LIN {X 0,Y 331.873,Z 625.786,A -85,B 0,C 180,E1 -14668.787,E2 -14668.787} C_VEL
LIN {X 0,Y 331.873,Z 625.82,A -85,B 0,C 180,E1 -14671.213,E2 -14671.213} C_VEL
LIN {X 0,Y 332.002,Z 624.514,A -85,B 0,C 180,E1 -14673.641,E2 -14673.641} C_VEL
LIN {X 0,Y 332.144,Z 621.851,A -85,B 0,C 180,E1 -14676.073,E2 -14676.073} C_VEL
LIN {X 0,Y 332.562,Z 617.761,A -85,B 0,C 180,E1 -14678.507,E2 -14678.507} C_VEL
LIN {X 0,Y 333.251,Z 612.118,A -85,B 0,C 180,E1 -14680.941,E2 -14680.941} C_VEL
LIN {X 0,Y 334.263,Z 605.737,A -85,B 0,C 180,E1 -14683.063,E2 -14683.063} C_VEL
LIN {X 0,Y 335.336,Z 598.598,A -85,B 0,C 180,E1 -14684.985,E2 -14684.985} C_VEL
LIN {X 0,Y 336.771,Z 589.501,A -85,B 0,C 180,E1 -14686.988,E2 -14686.988} C_VEL
LIN {X 0,Y 338.406,Z 579.466,A -85,B 0,C 180,E1 -14688.778,E2 -14688.778} C_VEL
LIN {X 0,Y 340.141,Z 568.232,A -85,B 0,C 180,E1 -14690.406,E2 -14690.406} C_VEL
LIN {X 0,Y 342.003,Z 555.922,A -85,B 0,C 180,E1 -14691.84,E2 -14691.84} C_VEL
LIN {X 0,Y 343.496,Z 543.513,A -85,B 0,C 180,E1 -14693.005,E2 -14693.005} C_VEL
LIN {X 0,Y 344.422,Z 532.816,A -85,B 0,C 180,E1 -14693.822,E2 -14693.822} C_VEL
LIN {X 0,Y 342.468,Z 519.71,A -85,B 0,C 180,E1 -14694.821,E2 -14694.821} C_VEL
LIN {X 0,Y 339.384,Z 505.28,A -85,B 0,C 180,E1 -14695.737,E2 -14695.737} C_VEL
LIN {X 0,Y 335.483,Z 491.266,A -85,B 0,C 180,E1 -14696.482,E2 -14696.482} C_VEL
LIN {X 0,Y 336.062,Z 480.841,A -85,B 0,C 180,E1 -14700.126,E2 -14700.126} C_VEL
LIN {X 0,Y 336.692,Z 470.956,A -85,B 0,C 180,E1 -14703.749,E2 -14703.749} C_VEL
LIN {X 0,Y 337.429,Z 460.368,A -85,B 0,C 180,E1 -14707.725,E2 -14707.725} C_VEL
LIN {X 0,Y 337.849,Z 455.305,A -85,B 0,C 180,E1 -14709.674,E2 -14709.674} C_VEL
LIN {X 0,Y 337.284,Z 449.99,A -85,B 0,C 180,E1 -14711.82,E2 -14711.82} C_VEL
LIN {X 0,Y 337.024,Z 448.414,A -85,B 0,C 180,E1 -14712.464,E2 -14712.464} C_VEL
LIN {X 0,Y 335.911,Z 446.445,A -85,B 0,C 180,E1 -14713.393,E2 -14713.393} C_VEL
LIN {X 0,Y 332.443,Z 443.786,A -85,B 0,C 180,E1 -14714.92,E2 -14714.92} C_VEL
LIN {X 0,Y 329.565,Z 441.699,A -85,B 0,C 180,E1 -14716.158,E2 -14716.158} C_VEL
LIN {X 0,Y 328.141,Z 439.808,A -85,B 0,C 180,E1 -14717.112,E2 -14717.112} C_VEL
LIN {X 0,Y 327.913,Z 439.09,A -85,B 0,C 180,E1 -14717.433,E2 -14717.433} C_VEL
LIN {X 0,Y 326.575,Z 433.434,A -85,B 0,C 180,E1 -14719.993,E2 -14719.993} C_VEL
LIN {X 0,Y 326.632,Z 433.419,A -85,B 0,C 180,E1 -14722.953,E2 -14722.953} C_VEL
LIN {X 0,Y 326.608,Z 433.417,A -85,B 0,C 180,E1 -14725.981,E2 -14725.981} C_VEL
LIN {X 0,Y 326.662,Z 433.41,A -85,B 0,C 180,E1 -14730.341,E2 -14730.341} C_VEL
LIN {X 0,Y 326.723,Z 433.414,A -85,B 0,C 180,E1 -14732.753,E2 -14732.753} C_VEL
LIN {X 0,Y 331.867,Z 449.308,A -85,B 0,C 180,E1 -14734.256,E2 -14734.256} C_VEL
LIN {X 0,Y 336.117,Z 463.308,A -85,B 0,C 180,E1 -14735.79,E2 -14735.79} C_VEL
LIN {X 0,Y 334.703,Z 476.843,A -85,B 0,C 180,E1 -14737.207,E2 -14737.207} C_VEL
LIN {X 0,Y 333.158,Z 489.7,A -85,B 0,C 180,E1 -14738.829,E2 -14738.829} C_VEL
LIN {X 0,Y 331.728,Z 500.872,A -85,B 0,C 180,E1 -14740.508,E2 -14740.508} C_VEL
LIN {X 0,Y 330.337,Z 511.243,A -85,B 0,C 180,E1 -14742.352,E2 -14742.352} C_VEL
LIN {X 0,Y 329.006,Z 521.51,A -85,B 0,C 180,E1 -14744.548,E2 -14744.548} C_VEL
LIN {X 0,Y 328.113,Z 528.711,A -85,B 0,C 180,E1 -14746.372,E2 -14746.372} C_VEL
LIN {X 0,Y 327.375,Z 534.919,A -85,B 0,C 180,E1 -14748.232,E2 -14748.232} C_VEL
LIN {X 0,Y 326.657,Z 541.736,A -85,B 0,C 180,E1 -14750.714,E2 -14750.714} C_VEL
LIN {X 0,Y 326.171,Z 547.048,A -85,B 0,C 180,E1 -14753.194,E2 -14753.194} C_VEL
LIN {X 0,Y 326.088,Z 550.153,A -85,B 0,C 180,E1 -14755.054,E2 -14755.054} C_VEL
LIN {X 0,Y 326.037,Z 551.802,A -85,B 0,C 180,E1 -14756.292,E2 -14756.292} C_VEL
LIN {X 0,Y 325.663,Z 554.196,A -85,B 0,C 180,E1 -14758.763,E2 -14758.763} C_VEL
LIN {X 0,Y 325.695,Z 555.343,A -85,B 0,C 180,E1 -14761.236,E2 -14761.236} C_VEL
LIN {X 0,Y 326.126,Z 555.262,A -85,B 0,C 180,E1 -14763.707,E2 -14763.707} C_VEL
LIN {X 0,Y 326.85,Z 553.984,A -85,B 0,C 180,E1 -14766.172,E2 -14766.172} C_VEL
LIN {X 0,Y 327.566,Z 551.529,A -85,B 0,C 180,E1 -14768.638,E2 -14768.638} C_VEL
LIN {X 0,Y 328.631,Z 547.803,A -85,B 0,C 180,E1 -14771.097,E2 -14771.097} C_VEL
LIN {X 0,Y 329.899,Z 542.755,A -85,B 0,C 180,E1 -14773.553,E2 -14773.553} C_VEL
LIN {X 0,Y 331.726,Z 536.167,A -85,B 0,C 180,E1 -14775.987,E2 -14775.987} C_VEL
LIN {X 0,Y 333.332,Z 530.273,A -85,B 0,C 180,E1 -14777.767,E2 -14777.767} C_VEL
LIN {X 0,Y 335.53,Z 521.743,A -85,B 0,C 180,E1 -14779.899,E2 -14779.899} C_VEL
LIN {X 0,Y 337.941,Z 511.714,A -85,B 0,C 180,E1 -14781.983,E2 -14781.983} C_VEL
LIN {X 0,Y 340.369,Z 501.358,A -85,B 0,C 180,E1 -14783.743,E2 -14783.743} C_VEL
LIN {X 0,Y 342.799,Z 490.786,A -85,B 0,C 180,E1 -14785.247,E2 -14785.247} C_VEL
LIN {X 0,Y 345.29,Z 477.829,A -85,B 0,C 180,E1 -14786.809,E2 -14786.809} C_VEL
LIN {X 0,Y 345.923,Z 474.416,A -85,B 0,C 180,E1 -14787.17,E2 -14787.17} C_VEL
LIN {X 0,Y 345.625,Z 471.773,A -85,B 0,C 180,E1 -14787.571,E2 -14787.571} C_VEL
LIN {X 0,Y 342.511,Z 461.947,A -85,B 0,C 180,E1 -14789.341,E2 -14789.341} C_VEL
LIN {X 0,Y 338.653,Z 453.425,A -85,B 0,C 180,E1 -14791.112,E2 -14791.112} C_VEL
LIN {X 0,Y 335.334,Z 447.304,A -85,B 0,C 180,E1 -14792.574,E2 -14792.574} C_VEL
LIN {X 0,Y 332.623,Z 443.026,A -85,B 0,C 180,E1 -14793.782,E2 -14793.782} C_VEL
LIN {X 0,Y 329.74,Z 438.96,A -85,B 0,C 180,E1 -14795.133,E2 -14795.133} C_VEL
LIN {X 0,Y 327.765,Z 437.307,A -85,B 0,C 180,E1 -14796.036,E2 -14796.036} C_VEL
LIN {X 0,Y 327.108,Z 435.891,A -85,B 0,C 180,E1 -14796.502,E2 -14796.502} C_VEL
LIN {X 0,Y 327.676,Z 439.473,A -85,B 0,C 180,E1 -14800.049,E2 -14800.049} C_VEL
LIN {X 0,Y 328.164,Z 442.306,A -85,B 0,C 180,E1 -14802.424,E2 -14802.424} C_VEL
LIN {X 0,Y 328.168,Z 444.668,A -85,B 0,C 180,E1 -14804.157,E2 -14804.157} C_VEL
LIN {X 0,Y 327.273,Z 451.1,A -85,B 0,C 180,E1 -14808.263,E2 -14808.263} C_VEL
LIN {X 0,Y 326.824,Z 457.809,A -85,B 0,C 180,E1 -14812.135,E2 -14812.135} C_VEL
LIN {X 0,Y 326.571,Z 463.902,A -85,B 0,C 180,E1 -14815.413,E2 -14815.413} C_VEL
LIN {X 0,Y 326.57,Z 464.705,A -85,B 0,C 180,E1 -14815.695,E2 -14815.695} C_VEL
LIN {X 0,Y 327.406,Z 468.646,A -85,B 0,C 180,E1 -14816.306,E2 -14816.306} C_VEL
LIN {X 0,Y 329.147,Z 472.574,A -85,B 0,C 180,E1 -14817.115,E2 -14817.115} C_VEL
LIN {X 0,Y 330.081,Z 476.56,A -85,B 0,C 180,E1 -14817.691,E2 -14817.691} C_VEL
LIN {X 0,Y 331.041,Z 478.958,A -85,B 0,C 180,E1 -14818.125,E2 -14818.125} C_VEL
LIN {X 0,Y 332.455,Z 484.387,A -85,B 0,C 180,E1 -14818.908,E2 -14818.908} C_VEL
LIN {X 0,Y 334.889,Z 495.067,A -85,B 0,C 180,E1 -14820.344,E2 -14820.344} C_VEL
LIN {X 0,Y 336.866,Z 508.787,A -85,B 0,C 180,E1 -14821.993,E2 -14821.993} C_VEL
LIN {X 0,Y 337.451,Z 521.179,A -85,B 0,C 180,E1 -14823.4,E2 -14823.4} C_VEL
LIN {X 0,Y 336.728,Z 537.938,A -85,B 0,C 180,E1 -14825.328,E2 -14825.328} C_VEL
LIN {X 0,Y 336.663,Z 546.487,A -85,B 0,C 180,E1 -14826.469,E2 -14826.469} C_VEL
LIN {X 0,Y 335.948,Z 551.732,A -85,B 0,C 180,E1 -14826.961,E2 -14826.961} C_VEL
LIN {X 0,Y 334.463,Z 563.284,A -85,B 0,C 180,E1 -14828.101,E2 -14828.101} C_VEL
LIN {X 0,Y 332.625,Z 575.509,A -85,B 0,C 180,E1 -14829.597,E2 -14829.597} C_VEL
LIN {X 0,Y 331.031,Z 585.559,A -85,B 0,C 180,E1 -14831.109,E2 -14831.109} C_VEL
LIN {X 0,Y 329.359,Z 595.531,A -85,B 0,C 180,E1 -14832.938,E2 -14832.938} C_VEL
LIN {X 0,Y 328.18,Z 603.43,A -85,B 0,C 180,E1 -14834.697,E2 -14834.697} C_VEL
LIN {X 0,Y 326.9,Z 611.673,A -85,B 0,C 180,E1 -14836.954,E2 -14836.954} C_VEL
LIN {X 0,Y 326.037,Z 617.186,A -85,B 0,C 180,E1 -14838.814,E2 -14838.814} C_VEL
LIN {X 0,Y 325.388,Z 622.949,A -85,B 0,C 180,E1 -14841.304,E2 -14841.304} C_VEL
LIN {X 0,Y 325.053,Z 627.131,A -85,B 0,C 180,E1 -14843.794,E2 -14843.794} C_VEL
LIN {X 0,Y 324.937,Z 629.863,A -85,B 0,C 180,E1 -14846.28,E2 -14846.28} C_VEL
LIN {X 0,Y 324.857,Z 631.218,A -85,B 0,C 180,E1 -14848.76,E2 -14848.76} C_VEL
LIN {X 0,Y 324.857,Z 631.216,A -85,B 0,C 180,E1 -14851.24,E2 -14851.24} C_VEL
LIN {X 0,Y 324.932,Z 629.857,A -85,B 0,C 180,E1 -14853.72,E2 -14853.72} C_VEL
LIN {X 0,Y 325.011,Z 627.122,A -85,B 0,C 180,E1 -14856.207,E2 -14856.207} C_VEL
LIN {X 0,Y 325.382,Z 622.931,A -85,B 0,C 180,E1 -14858.696,E2 -14858.696} C_VEL
LIN {X 0,Y 326.029,Z 617.159,A -85,B 0,C 180,E1 -14861.187,E2 -14861.187} C_VEL
LIN {X 0,Y 327.059,Z 610.636,A -85,B 0,C 180,E1 -14863.356,E2 -14863.356} C_VEL
LIN {X 0,Y 328.14,Z 602.769,A -85,B 0,C 180,E1 -14865.464,E2 -14865.464} C_VEL
LIN {X 0,Y 329.609,Z 593.978,A -85,B 0,C 180,E1 -14867.368,E2 -14867.368} C_VEL
LIN {X 0,Y 331.256,Z 583.611,A -85,B 0,C 180,E1 -14869.199,E2 -14869.199} C_VEL
LIN {X 0,Y 332.951,Z 573.163,A -85,B 0,C 180,E1 -14870.705,E2 -14870.705} C_VEL
LIN {X 0,Y 334.638,Z 561.769,A -85,B 0,C 180,E1 -14872.049,E2 -14872.049} C_VEL
LIN {X 0,Y 336.113,Z 549.889,A -85,B 0,C 180,E1 -14873.186,E2 -14873.186} C_VEL
LIN {X 0,Y 336.405,Z 544.502,A -85,B 0,C 180,E1 -14873.647,E2 -14873.647} C_VEL
LIN {X 0,Y 334.969,Z 531.463,A -85,B 0,C 180,E1 -14874.731,E2 -14874.731} C_VEL
LIN {X 0,Y 332.626,Z 516.987,A -85,B 0,C 180,E1 -14875.72,E2 -14875.72} C_VEL
LIN {X 0,Y 329.791,Z 502.321,A -85,B 0,C 180,E1 -14876.487,E2 -14876.487} C_VEL
LIN {X 0,Y 326.806,Z 490.048,A -85,B 0,C 180,E1 -14877.048,E2 -14877.048} C_VEL
LIN {X 0,Y 326.391,Z 486.716,A -85,B 0,C 180,E1 -14877.491,E2 -14877.491} C_VEL
LIN {X 0,Y 326.933,Z 480.059,A -85,B 0,C 180,E1 -14881.059,E2 -14881.059} C_VEL
LIN {X 0,Y 327.472,Z 473.478,A -85,B 0,C 180,E1 -14884.646,E2 -14884.646} C_VEL
LIN {X 0,Y 327.976,Z 466.679,A -85,B 0,C 180,E1 -14888.42,E2 -14888.42} C_VEL
LIN {X 0,Y 328.616,Z 459.795,A -85,B 0,C 180,E1 -14892.352,E2 -14892.352} C_VEL
LIN {X 0,Y 329.189,Z 453.882,A -85,B 0,C 180,E1 -14895.805,E2 -14895.805} C_VEL
LIN {X 0,Y 329.373,Z 449.755,A -85,B 0,C 180,E1 -14898.315,E2 -14898.315} C_VEL
LIN {X 0,Y 328.587,Z 444.529,A -85,B 0,C 180,E1 -14901.664,E2 -14901.664} C_VEL
LIN {X 0,Y 327.61,Z 439.041,A -85,B 0,C 180,E1 -14905.355,E2 -14905.355} C_VEL
LIN {X 0,Y 326.68,Z 433.42,A -85,B 0,C 180,E1 -14909.377,E2 -14909.377} C_VEL
LIN {X 0,Y 326.686,Z 433.404,A -85,B 0,C 180,E1 -14913.143,E2 -14913.143} C_VEL
LIN {X 0,Y 326.653,Z 433.419,A -85,B 0,C 180,E1 -14915.871,E2 -14915.871} C_VEL
LIN {X 0,Y 326.666,Z 433.402,A -85,B 0,C 180,E1 -14919.865,E2 -14919.865} C_VEL
LIN {X 0,Y 326.701,Z 433.415,A -85,B 0,C 180,E1 -14922.472,E2 -14922.472} C_VEL
LIN {X 0,Y 326.761,Z 433.396,A -85,B 0,C 180,E1 -14926.315,E2 -14926.315} C_VEL
LIN {X 0,Y 326.785,Z 433.391,A -85,B 0,C 180,E1 -14930.093,E2 -14930.093} C_VEL
LIN {X 0,Y 326.985,Z 433.38,A -85,B 0,C 180,E1 -14933.831,E2 -14933.831} C_VEL
LIN {X 0,Y 327.048,Z 433.354,A -85,B 0,C 180,E1 -14937.537,E2 -14937.537} C_VEL
LIN {X 0,Y 327.219,Z 433.353,A -85,B 0,C 180,E1 -14940,E2 -14940} C_VEL
LIN {X 0,Y 327.047,Z 433.356,A -85,B 0,C 180,E1 -14942.463,E2 -14942.463} C_VEL
LIN {X 0,Y 326.973,Z 433.375,A -85,B 0,C 180,E1 -14946.665,E2 -14946.665} C_VEL
LIN {X 0,Y 326.816,Z 433.394,A -85,B 0,C 180,E1 -14949.906,E2 -14949.906} C_VEL
LIN {X 0,Y 326.761,Z 433.394,A -85,B 0,C 180,E1 -14953.685,E2 -14953.685} C_VEL
LIN {X 0,Y 326.701,Z 433.41,A -85,B 0,C 180,E1 -14957.528,E2 -14957.528} C_VEL
LIN {X 0,Y 326.66,Z 433.42,A -85,B 0,C 180,E1 -14960.135,E2 -14960.135} C_VEL
LIN {X 0,Y 326.651,Z 433.418,A -85,B 0,C 180,E1 -14964.129,E2 -14964.129} C_VEL
LIN {X 0,Y 326.686,Z 433.408,A -85,B 0,C 180,E1 -14966.858,E2 -14966.858} C_VEL
LIN {X 0,Y 326.64,Z 433.418,A -85,B 0,C 180,E1 -14970.611,E2 -14970.611} C_VEL
LIN {X 0,Y 326.608,Z 433.427,A -85,B 0,C 180,E1 -14974.019,E2 -14974.019} C_VEL
LIN {X 0,Y 326.629,Z 433.424,A -85,B 0,C 180,E1 -14977.239,E2 -14977.239} C_VEL
LIN {X 0,Y 326.591,Z 433.465,A -85,B 0,C 180,E1 -14980.209,E2 -14980.209} C_VEL
LIN {X 0,Y 328.202,Z 440.412,A -85,B 0,C 180,E1 -14983.276,E2 -14983.276} C_VEL
LIN {X 0,Y 329.71,Z 447.69,A -85,B 0,C 180,E1 -14986.447,E2 -14986.447} C_VEL
LIN {X 0,Y 330.874,Z 454.772,A -85,B 0,C 180,E1 -14989.421,E2 -14989.421} C_VEL
LIN {X 0,Y 330.831,Z 459.25,A -85,B 0,C 180,E1 -14991.195,E2 -14991.195} C_VEL
LIN {X 0,Y 330.039,Z 468.945,A -85,B 0,C 180,E1 -14994.904,E2 -14994.904} C_VEL
LIN {X 0,Y 329.393,Z 478.804,A -85,B 0,C 180,E1 -14998.589,E2 -14998.589} C_VEL
LIN {X 0,Y 328.709,Z 489.231,A -85,B 0,C 180,E1 -15002.323,E2 -15002.323} C_VEL
LIN {X 0,Y 328.622,Z 491.3,A -85,B 0,C 180,E1 -15003.043,E2 -15003.043} C_VEL
LIN {X 0,Y 333.181,Z 507.767,A -85,B 0,C 180,E1 -15003.955,E2 -15003.955} C_VEL
LIN {X 0,Y 335.987,Z 521.344,A -85,B 0,C 180,E1 -15004.867,E2 -15004.867} C_VEL
LIN {X 0,Y 337.83,Z 534.358,A -85,B 0,C 180,E1 -15005.904,E2 -15005.904} C_VEL
LIN {X 0,Y 336.477,Z 547.218,A -85,B 0,C 180,E1 -15006.942,E2 -15006.942} C_VEL
LIN {X 0,Y 334.927,Z 558.972,A -85,B 0,C 180,E1 -15008.133,E2 -15008.133} C_VEL
LIN {X 0,Y 333.02,Z 570.868,A -85,B 0,C 180,E1 -15009.622,E2 -15009.622} C_VEL
LIN {X 0,Y 331.469,Z 580.723,A -85,B 0,C 180,E1 -15011.135,E2 -15011.135} C_VEL
LIN {X 0,Y 329.748,Z 590.533,A -85,B 0,C 180,E1 -15012.959,E2 -15012.959} C_VEL
LIN {X 0,Y 328.425,Z 598.615,A -85,B 0,C 180,E1 -15014.787,E2 -15014.787} C_VEL
LIN {X 0,Y 327.375,Z 605.463,A -85,B 0,C 180,E1 -15016.657,E2 -15016.657} C_VEL
LIN {X 0,Y 326.307,Z 611.907,A -85,B 0,C 180,E1 -15018.823,E2 -15018.823} C_VEL
LIN {X 0,Y 325.516,Z 617.615,A -85,B 0,C 180,E1 -15021.307,E2 -15021.307} C_VEL
LIN {X 0,Y 325.112,Z 621.765,A -85,B 0,C 180,E1 -15023.795,E2 -15023.795} C_VEL
LIN {X 0,Y 324.911,Z 624.482,A -85,B 0,C 180,E1 -15026.279,E2 -15026.279} C_VEL
LIN {X 0,Y 324.785,Z 625.845,A -85,B 0,C 180,E1 -15028.76,E2 -15028.76} C_VEL
LIN {X 0,Y 324.785,Z 625.878,A -85,B 0,C 180,E1 -15031.24,E2 -15031.24} C_VEL
LIN {X 0,Y 324.909,Z 624.572,A -85,B 0,C 180,E1 -15033.721,E2 -15033.721} C_VEL
LIN {X 0,Y 325.078,Z 621.908,A -85,B 0,C 180,E1 -15036.206,E2 -15036.206} C_VEL
LIN {X 0,Y 325.513,Z 617.818,A -85,B 0,C 180,E1 -15038.693,E2 -15038.693} C_VEL
LIN {X 0,Y 326.252,Z 612.173,A -85,B 0,C 180,E1 -15041.179,E2 -15041.179} C_VEL
LIN {X 0,Y 327.332,Z 605.791,A -85,B 0,C 180,E1 -15043.345,E2 -15043.345} C_VEL
LIN {X 0,Y 328.407,Z 598.891,A -85,B 0,C 180,E1 -15045.246,E2 -15045.246} C_VEL
LIN {X 0,Y 329.959,Z 589.552,A -85,B 0,C 180,E1 -15047.349,E2 -15047.349} C_VEL
LIN {X 0,Y 331.674,Z 579.513,A -85,B 0,C 180,E1 -15049.174,E2 -15049.174} C_VEL
LIN {X 0,Y 333.49,Z 568.275,A -85,B 0,C 180,E1 -15050.832,E2 -15050.832} C_VEL
LIN {X 0,Y 335.406,Z 556.051,A -85,B 0,C 180,E1 -15052.281,E2 -15052.281} C_VEL
LIN {X 0,Y 336.993,Z 543.216,A -85,B 0,C 180,E1 -15053.506,E2 -15053.506} C_VEL
LIN {X 0,Y 337.882,Z 534.69,A -85,B 0,C 180,E1 -15054.174,E2 -15054.174} C_VEL
LIN {X 0,Y 336.07,Z 521.646,A -85,B 0,C 180,E1 -15055.217,E2 -15055.217} C_VEL
LIN {X 0,Y 333.145,Z 507.533,A -85,B 0,C 180,E1 -15056.165,E2 -15056.165} C_VEL
LIN {X 0,Y 328.615,Z 491.257,A -85,B 0,C 180,E1 -15057.082,E2 -15057.082} C_VEL
LIN {X 0,Y 329.268,Z 480.763,A -85,B 0,C 180,E1 -15060.815,E2 -15060.815} C_VEL
LIN {X 0,Y 329.91,Z 471.177,A -85,B 0,C 180,E1 -15064.369,E2 -15064.369} C_VEL
LIN {X 0,Y 330.635,Z 461.278,A -85,B 0,C 180,E1 -15068.142,E2 -15068.142} C_VEL
LIN {X 0,Y 330.991,Z 456.139,A -85,B 0,C 180,E1 -15070.146,E2 -15070.146} C_VEL
LIN {X 0,Y 330.219,Z 450.389,A -85,B 0,C 180,E1 -15072.539,E2 -15072.539} C_VEL
LIN {X 0,Y 328.665,Z 442.467,A -85,B 0,C 180,E1 -15075.976,E2 -15075.976} C_VEL
LIN {X 0,Y 327.913,Z 439.09,A -85,B 0,C 180,E1 -15077.433,E2 -15077.433} C_VEL
LIN {X 0,Y 326.906,Z 437.972,A -85,B 0,C 180,E1 -15078.065,E2 -15078.065} C_VEL
LIN {X 0,Y 320.343,Z 435.415,A -85,B 0,C 180,E1 -15080.099,E2 -15080.099} C_VEL
LIN {X 0,Y 319.592,Z 434.302,A -85,B 0,C 180,E1 -15080.798,E2 -15080.798} C_VEL
LIN {X 0,Y 319.582,Z 434.304,A -85,B 0,C 180,E1 -15084.457,E2 -15084.457} C_VEL
LIN {X 0,Y 319.534,Z 434.308,A -85,B 0,C 180,E1 -15088.138,E2 -15088.138} C_VEL
LIN {X 0,Y 319.646,Z 434.295,A -85,B 0,C 180,E1 -15091.924,E2 -15091.924} C_VEL
LIN {X 0,Y 319.662,Z 434.293,A -85,B 0,C 180,E1 -15092.359,E2 -15092.359} C_VEL
LIN {X 0,Y 324.546,Z 449.336,A -85,B 0,C 180,E1 -15093.804,E2 -15093.804} C_VEL
LIN {X 0,Y 328.56,Z 462.529,A -85,B 0,C 180,E1 -15095.261,E2 -15095.261} C_VEL
LIN {X 0,Y 329.266,Z 464.876,A -85,B 0,C 180,E1 -15095.543,E2 -15095.543} C_VEL
LIN {X 0,Y 327.815,Z 478.105,A -85,B 0,C 180,E1 -15096.967,E2 -15096.967} C_VEL
LIN {X 0,Y 326.322,Z 490.19,A -85,B 0,C 180,E1 -15098.523,E2 -15098.523} C_VEL
LIN {X 0,Y 324.694,Z 502.333,A -85,B 0,C 180,E1 -15100.397,E2 -15100.397} C_VEL
LIN {X 0,Y 323.285,Z 512.586,A -85,B 0,C 180,E1 -15102.281,E2 -15102.281} C_VEL
LIN {X 0,Y 322.057,Z 521.771,A -85,B 0,C 180,E1 -15104.28,E2 -15104.28} C_VEL
LIN {X 0,Y 321.032,Z 529.91,A -85,B 0,C 180,E1 -15106.388,E2 -15106.388} C_VEL
LIN {X 0,Y 320.184,Z 537.01,A -85,B 0,C 180,E1 -15108.606,E2 -15108.606} C_VEL
LIN {X 0,Y 319.479,Z 543.59,A -85,B 0,C 180,E1 -15111.142,E2 -15111.142} C_VEL
LIN {X 0,Y 319.043,Z 548.682,A -85,B 0,C 180,E1 -15113.676,E2 -15113.676} C_VEL
LIN {X 0,Y 318.972,Z 552.404,A -85,B 0,C 180,E1 -15116.21,E2 -15116.21} C_VEL
LIN {X 0,Y 318.621,Z 554.887,A -85,B 0,C 180,E1 -15118.736,E2 -15118.736} C_VEL
LIN {X 0,Y 318.651,Z 556.143,A -85,B 0,C 180,E1 -15121.264,E2 -15121.264} C_VEL
LIN {X 0,Y 319.104,Z 556.18,A -85,B 0,C 180,E1 -15123.788,E2 -15123.788} C_VEL
LIN {X 0,Y 319.864,Z 555.008,A -85,B 0,C 180,E1 -15126.307,E2 -15126.307} C_VEL
LIN {X 0,Y 320.651,Z 552.676,A -85,B 0,C 180,E1 -15128.825,E2 -15128.825} C_VEL
LIN {X 0,Y 321.788,Z 549.083,A -85,B 0,C 180,E1 -15131.336,E2 -15131.336} C_VEL
LIN {X 0,Y 323.138,Z 544.164,A -85,B 0,C 180,E1 -15133.842,E2 -15133.842} C_VEL
LIN {X 0,Y 325.08,Z 537.764,A -85,B 0,C 180,E1 -15136.323,E2 -15136.323} C_VEL
LIN {X 0,Y 326.812,Z 531.873,A -85,B 0,C 180,E1 -15138.169,E2 -15138.169} C_VEL
LIN {X 0,Y 329.128,Z 523.736,A -85,B 0,C 180,E1 -15140.303,E2 -15140.303} C_VEL
LIN {X 0,Y 331.678,Z 513.904,A -85,B 0,C 180,E1 -15142.421,E2 -15142.421} C_VEL
LIN {X 0,Y 334.25,Z 503.91,A -85,B 0,C 180,E1 -15144.205,E2 -15144.205} C_VEL
LIN {X 0,Y 337.181,Z 491.975,A -85,B 0,C 180,E1 -15145.958,E2 -15145.958} C_VEL
LIN {X 0,Y 339.535,Z 480.884,A -85,B 0,C 180,E1 -15147.343,E2 -15147.343} C_VEL
LIN {X 0,Y 340.297,Z 476.944,A -85,B 0,C 180,E1 -15147.785,E2 -15147.785} C_VEL
LIN {X 0,Y 339.688,Z 473.304,A -85,B 0,C 180,E1 -15148.415,E2 -15148.415} C_VEL
LIN {X 0,Y 337.096,Z 465.108,A -85,B 0,C 180,E1 -15150.024,E2 -15150.024} C_VEL
LIN {X 0,Y 333.288,Z 456.378,A -85,B 0,C 180,E1 -15152.019,E2 -15152.019} C_VEL
LIN {X 0,Y 329.76,Z 449.903,A -85,B 0,C 180,E1 -15153.779,E2 -15153.779} C_VEL
LIN {X 0,Y 326.968,Z 445.59,A -85,B 0,C 180,E1 -15155.235,E2 -15155.235} C_VEL
LIN {X 0,Y 325.259,Z 444.147,A -85,B 0,C 180,E1 -15156.081,E2 -15156.081} C_VEL
LIN {X 0,Y 324.266,Z 442.628,A -85,B 0,C 180,E1 -15156.686,E2 -15156.686} C_VEL
LIN {X 0,Y 322.352,Z 442.114,A -85,B 0,C 180,E1 -15157.623,E2 -15157.623} C_VEL
LIN {X 0,Y 320.756,Z 440.393,A -85,B 0,C 180,E1 -15158.788,E2 -15158.788} C_VEL
LIN {X 0,Y 320.593,Z 439.96,A -85,B 0,C 180,E1 -15159.023,E2 -15159.023} C_VEL
LIN {X 0,Y 321.153,Z 443.19,A -85,B 0,C 180,E1 -15161.923,E2 -15161.923} C_VEL
LIN {X 0,Y 321.126,Z 446.533,A -85,B 0,C 180,E1 -15164.454,E2 -15164.454} C_VEL
LIN {X 0,Y 320.211,Z 453.259,A -85,B 0,C 180,E1 -15168.819,E2 -15168.819} C_VEL
LIN {X 0,Y 319.734,Z 460.23,A -85,B 0,C 180,E1 -15172.901,E2 -15172.901} C_VEL
LIN {X 0,Y 320.468,Z 464.183,A -85,B 0,C 180,E1 -15173.692,E2 -15173.692} C_VEL
LIN {X 0,Y 322.63,Z 469.537,A -85,B 0,C 180,E1 -15175.048,E2 -15175.048} C_VEL
LIN {X 0,Y 323.754,Z 474.413,A -85,B 0,C 180,E1 -15175.904,E2 -15175.904} C_VEL
LIN {X 0,Y 324.916,Z 477.501,A -85,B 0,C 180,E1 -15176.551,E2 -15176.551} C_VEL
LIN {X 0,Y 328.151,Z 490.791,A -85,B 0,C 180,E1 -15178.675,E2 -15178.675} C_VEL
LIN {X 0,Y 330.201,Z 502.399,A -85,B 0,C 180,E1 -15180.292,E2 -15180.292} C_VEL
LIN {X 0,Y 331.337,Z 514.643,A -85,B 0,C 180,E1 -15181.829,E2 -15181.829} C_VEL
LIN {X 0,Y 331.319,Z 525.862,A -85,B 0,C 180,E1 -15183.172,E2 -15183.172} C_VEL
LIN {X 0,Y 330.324,Z 541.724,A -85,B 0,C 180,E1 -15185.153,E2 -15185.153} C_VEL
LIN {X 0,Y 330.235,Z 547.509,A -85,B 0,C 180,E1 -15185.983,E2 -15185.983} C_VEL
LIN {X 0,Y 329.531,Z 550.892,A -85,B 0,C 180,E1 -15186.407,E2 -15186.407} C_VEL
LIN {X 0,Y 327.853,Z 563.245,A -85,B 0,C 180,E1 -15187.636,E2 -15187.636} C_VEL
LIN {X 0,Y 325.962,Z 575.463,A -85,B 0,C 180,E1 -15189.16,E2 -15189.16} C_VEL
LIN {X 0,Y 324.295,Z 585.511,A -85,B 0,C 180,E1 -15190.701,E2 -15190.701} C_VEL
LIN {X 0,Y 322.552,Z 595.48,A -85,B 0,C 180,E1 -15192.567,E2 -15192.567} C_VEL
LIN {X 0,Y 321.209,Z 603.891,A -85,B 0,C 180,E1 -15194.493,E2 -15194.493} C_VEL
LIN {X 0,Y 319.954,Z 611.618,A -85,B 0,C 180,E1 -15196.665,E2 -15196.665} C_VEL
LIN {X 0,Y 319.025,Z 617.13,A -85,B 0,C 180,E1 -15198.564,E2 -15198.564} C_VEL
LIN {X 0,Y 318.347,Z 622.893,A -85,B 0,C 180,E1 -15201.11,E2 -15201.11} C_VEL
LIN {X 0,Y 317.971,Z 627.074,A -85,B 0,C 180,E1 -15203.655,E2 -15203.655} C_VEL
LIN {X 0,Y 317.845,Z 629.805,A -85,B 0,C 180,E1 -15206.197,E2 -15206.197} C_VEL
LIN {X 0,Y 317.768,Z 631.16,A -85,B 0,C 180,E1 -15208.733,E2 -15208.733} C_VEL
LIN {X 0,Y 317.768,Z 631.157,A -85,B 0,C 180,E1 -15211.267,E2 -15211.267} C_VEL
LIN {X 0,Y 317.839,Z 629.799,A -85,B 0,C 180,E1 -15213.804,E2 -15213.804} C_VEL
LIN {X 0,Y 317.951,Z 627.063,A -85,B 0,C 180,E1 -15216.345,E2 -15216.345} C_VEL
LIN {X 0,Y 318.341,Z 622.872,A -85,B 0,C 180,E1 -15218.89,E2 -15218.89} C_VEL
LIN {X 0,Y 319.018,Z 617.101,A -85,B 0,C 180,E1 -15221.436,E2 -15221.436} C_VEL
LIN {X 0,Y 320.121,Z 610.579,A -85,B 0,C 180,E1 -15223.651,E2 -15223.651} C_VEL
LIN {X 0,Y 321.354,Z 602.335,A -85,B 0,C 180,E1 -15225.894,E2 -15225.894} C_VEL
LIN {X 0,Y 322.803,Z 593.922,A -85,B 0,C 180,E1 -15227.746,E2 -15227.746} C_VEL
LIN {X 0,Y 324.54,Z 583.557,A -85,B 0,C 180,E1 -15229.613,E2 -15229.613} C_VEL
LIN {X 0,Y 326.297,Z 573.112,A -85,B 0,C 180,E1 -15231.148,E2 -15231.148} C_VEL
LIN {X 0,Y 328.053,Z 561.721,A -85,B 0,C 180,E1 -15232.516,E2 -15232.516} C_VEL
LIN {X 0,Y 329.564,Z 550.129,A -85,B 0,C 180,E1 -15233.648,E2 -15233.648} C_VEL
LIN {X 0,Y 329.827,Z 546.096,A -85,B 0,C 180,E1 -15234.009,E2 -15234.009} C_VEL
LIN {X 0,Y 328.492,Z 533.124,A -85,B 0,C 180,E1 -15235.142,E2 -15235.142} C_VEL
LIN {X 0,Y 326.242,Z 518.571,A -85,B 0,C 180,E1 -15236.185,E2 -15236.185} C_VEL
LIN {X 0,Y 323.421,Z 503.738,A -85,B 0,C 180,E1 -15237.009,E2 -15237.009} C_VEL
LIN {X 0,Y 320.854,Z 492.766,A -85,B 0,C 180,E1 -15237.527,E2 -15237.527} C_VEL
LIN {X 0,Y 319.931,Z 489.497,A -85,B 0,C 180,E1 -15237.719,E2 -15237.719} C_VEL
LIN {X 0,Y 319.409,Z 485.41,A -85,B 0,C 180,E1 -15238.342,E2 -15238.342} C_VEL
LIN {X 0,Y 319.909,Z 479.077,A -85,B 0,C 180,E1 -15241.82,E2 -15241.82} C_VEL
LIN {X 0,Y 320.411,Z 473.776,A -85,B 0,C 180,E1 -15244.771,E2 -15244.771} C_VEL
LIN {X 0,Y 320.937,Z 467.017,A -85,B 0,C 180,E1 -15248.625,E2 -15248.625} C_VEL
LIN {X 0,Y 321.611,Z 460.087,A -85,B 0,C 180,E1 -15252.643,E2 -15252.643} C_VEL
LIN {X 0,Y 322.195,Z 454.433,A -85,B 0,C 180,E1 -15256.04,E2 -15256.04} C_VEL
LIN {X 0,Y 322.318,Z 450.458,A -85,B 0,C 180,E1 -15258.495,E2 -15258.495} C_VEL
LIN {X 0,Y 321.857,Z 447.033,A -85,B 0,C 180,E1 -15260.711,E2 -15260.711} C_VEL
LIN {X 0,Y 320.942,Z 441.996,A -85,B 0,C 180,E1 -15264.118,E2 -15264.118} C_VEL
LIN {X 0,Y 319.938,Z 436.268,A -85,B 0,C 180,E1 -15268.183,E2 -15268.183} C_VEL
LIN {X 0,Y 319.633,Z 434.299,A -85,B 0,C 180,E1 -15269.712,E2 -15269.712} C_VEL
LIN {X 0,Y 319.636,Z 434.278,A -85,B 0,C 180,E1 -15273.912,E2 -15273.912} C_VEL
LIN {X 0,Y 319.598,Z 434.292,A -85,B 0,C 180,E1 -15278.048,E2 -15278.048} C_VEL
LIN {X 0,Y 319.691,Z 434.282,A -85,B 0,C 180,E1 -15280.962,E2 -15280.962} C_VEL
LIN {X 0,Y 319.732,Z 434.264,A -85,B 0,C 180,E1 -15285.276,E2 -15285.276} C_VEL
LIN {X 0,Y 319.717,Z 434.284,A -85,B 0,C 180,E1 -15288.59,E2 -15288.59} C_VEL
LIN {X 0,Y 319.896,Z 434.252,A -85,B 0,C 180,E1 -15292.425,E2 -15292.425} C_VEL
LIN {X 0,Y 319.746,Z 434.28,A -85,B 0,C 180,E1 -15294.956,E2 -15294.956} C_VEL
LIN {X 0,Y 319.991,Z 434.232,A -85,B 0,C 180,E1 -15297.483,E2 -15297.483} C_VEL
LIN {X 0,Y 320.17,Z 434.231,A -85,B 0,C 180,E1 -15300,E2 -15300} C_VEL
LIN {X 0,Y 319.991,Z 434.234,A -85,B 0,C 180,E1 -15302.518,E2 -15302.518} C_VEL
LIN {X 0,Y 319.933,Z 434.253,A -85,B 0,C 180,E1 -15306.656,E2 -15306.656} C_VEL
LIN {X 0,Y 319.76,Z 434.275,A -85,B 0,C 180,E1 -15310.127,E2 -15310.127} C_VEL
LIN {X 0,Y 319.732,Z 434.274,A -85,B 0,C 180,E1 -15314.724,E2 -15314.724} C_VEL
LIN {X 0,Y 319.69,Z 434.277,A -85,B 0,C 180,E1 -15319.038,E2 -15319.038} C_VEL
LIN {X 0,Y 319.562,Z 434.295,A -85,B 0,C 180,E1 -15323.32,E2 -15323.32} C_VEL
LIN {X 0,Y 319.636,Z 434.289,A -85,B 0,C 180,E1 -15326.088,E2 -15326.088} C_VEL
LIN {X 0,Y 319.591,Z 434.3,A -85,B 0,C 180,E1 -15328.934,E2 -15328.934} C_VEL
LIN {X 0,Y 319.534,Z 434.309,A -85,B 0,C 180,E1 -15331.862,E2 -15331.862} C_VEL
LIN {X 0,Y 319.581,Z 434.298,A -85,B 0,C 180,E1 -15335.543,E2 -15335.543} C_VEL
LIN {X 0,Y 319.576,Z 434.444,A -85,B 0,C 180,E1 -15339.489,E2 -15339.489} C_VEL
LIN {X 0,Y 321.222,Z 441.511,A -85,B 0,C 180,E1 -15342.707,E2 -15342.707} C_VEL
LIN {X 0,Y 322.726,Z 448.775,A -85,B 0,C 180,E1 -15345.943,E2 -15345.943} C_VEL
LIN {X 0,Y 323.834,Z 454.836,A -85,B 0,C 180,E1 -15348.554,E2 -15348.554} C_VEL
LIN {X 0,Y 324.113,Z 458.867,A -85,B 0,C 180,E1 -15350.233,E2 -15350.233} C_VEL
LIN {X 0,Y 323.317,Z 468.701,A -85,B 0,C 180,E1 -15354.062,E2 -15354.062} C_VEL
LIN {X 0,Y 322.614,Z 478.254,A -85,B 0,C 180,E1 -15357.688,E2 -15357.688} C_VEL
LIN {X 0,Y 321.971,Z 488.128,A -85,B 0,C 180,E1 -15361.3,E2 -15361.3} C_VEL
LIN {X 0,Y 321.794,Z 491.392,A -85,B 0,C 180,E1 -15362.432,E2 -15362.432} C_VEL
LIN {X 0,Y 326.317,Z 507.497,A -85,B 0,C 180,E1 -15363.354,E2 -15363.354} C_VEL
LIN {X 0,Y 329.09,Z 520.467,A -85,B 0,C 180,E1 -15364.25,E2 -15364.25} C_VEL
LIN {X 0,Y 331.012,Z 533.387,A -85,B 0,C 180,E1 -15365.298,E2 -15365.298} C_VEL
LIN {X 0,Y 331.135,Z 536.489,A -85,B 0,C 180,E1 -15365.557,E2 -15365.557} C_VEL
LIN {X 0,Y 329.768,Z 548.919,A -85,B 0,C 180,E1 -15366.62,E2 -15366.62} C_VEL
LIN {X 0,Y 327.983,Z 561.558,A -85,B 0,C 180,E1 -15367.976,E2 -15367.976} C_VEL
LIN {X 0,Y 326.007,Z 573.018,A -85,B 0,C 180,E1 -15369.493,E2 -15369.493} C_VEL
LIN {X 0,Y 324.423,Z 582.528,A -85,B 0,C 180,E1 -15371.038,E2 -15371.038} C_VEL
LIN {X 0,Y 322.668,Z 592.051,A -85,B 0,C 180,E1 -15372.9,E2 -15372.9} C_VEL
LIN {X 0,Y 321.336,Z 599.946,A -85,B 0,C 180,E1 -15374.784,E2 -15374.784} C_VEL
LIN {X 0,Y 320.253,Z 606.514,A -85,B 0,C 180,E1 -15376.678,E2 -15376.678} C_VEL
LIN {X 0,Y 319.316,Z 611.966,A -85,B 0,C 180,E1 -15378.575,E2 -15378.575} C_VEL
LIN {X 0,Y 318.482,Z 617.673,A -85,B 0,C 180,E1 -15381.114,E2 -15381.114} C_VEL
LIN {X 0,Y 318.054,Z 621.824,A -85,B 0,C 180,E1 -15383.657,E2 -15383.657} C_VEL
LIN {X 0,Y 317.822,Z 624.541,A -85,B 0,C 180,E1 -15386.196,E2 -15386.196} C_VEL
LIN {X 0,Y 317.699,Z 625.903,A -85,B 0,C 180,E1 -15388.732,E2 -15388.732} C_VEL
LIN {X 0,Y 317.699,Z 625.936,A -85,B 0,C 180,E1 -15391.268,E2 -15391.268} C_VEL
LIN {X 0,Y 317.819,Z 624.63,A -85,B 0,C 180,E1 -15393.804,E2 -15393.804} C_VEL
LIN {X 0,Y 318.012,Z 621.966,A -85,B 0,C 180,E1 -15396.344,E2 -15396.344} C_VEL
LIN {X 0,Y 318.479,Z 617.875,A -85,B 0,C 180,E1 -15398.886,E2 -15398.886} C_VEL
LIN {X 0,Y 319.237,Z 612.229,A -85,B 0,C 180,E1 -15401.428,E2 -15401.428} C_VEL
LIN {X 0,Y 320.38,Z 605.846,A -85,B 0,C 180,E1 -15403.64,E2 -15403.64} C_VEL
LIN {X 0,Y 321.698,Z 598.031,A -85,B 0,C 180,E1 -15405.817,E2 -15405.817} C_VEL
LIN {X 0,Y 323.157,Z 589.603,A -85,B 0,C 180,E1 -15407.726,E2 -15407.726} C_VEL
LIN {X 0,Y 324.957,Z 579.56,A -85,B 0,C 180,E1 -15409.586,E2 -15409.586} C_VEL
LIN {X 0,Y 326.852,Z 568.318,A -85,B 0,C 180,E1 -15411.275,E2 -15411.275} C_VEL
LIN {X 0,Y 328.672,Z 557.146,A -85,B 0,C 180,E1 -15412.637,E2 -15412.637} C_VEL
LIN {X 0,Y 330.261,Z 544.963,A -85,B 0,C 180,E1 -15413.849,E2 -15413.849} C_VEL
LIN {X 0,Y 331.297,Z 535.754,A -85,B 0,C 180,E1 -15414.602,E2 -15414.602} C_VEL
LIN {X 0,Y 329.585,Z 523.164,A -85,B 0,C 180,E1 -15415.658,E2 -15415.658} C_VEL
LIN {X 0,Y 326.722,Z 509.013,A -85,B 0,C 180,E1 -15416.659,E2 -15416.659} C_VEL
LIN {X 0,Y 322.504,Z 493.892,A -85,B 0,C 180,E1 -15417.551,E2 -15417.551} C_VEL
LIN {X 0,Y 321.792,Z 491.276,A -85,B 0,C 180,E1 -15417.696,E2 -15417.696} C_VEL
LIN {X 0,Y 322.336,Z 482.59,A -85,B 0,C 180,E1 -15420.822,E2 -15420.822} C_VEL
LIN {X 0,Y 323.012,Z 472.884,A -85,B 0,C 180,E1 -15424.451,E2 -15424.451} C_VEL
LIN {X 0,Y 323.893,Z 462.065,A -85,B 0,C 180,E1 -15428.634,E2 -15428.634} C_VEL
LIN {X 0,Y 324.11,Z 457.213,A -85,B 0,C 180,E1 -15430.581,E2 -15430.581} C_VEL
LIN {X 0,Y 323.177,Z 451.017,A -85,B 0,C 180,E1 -15433.238,E2 -15433.238} C_VEL
LIN {X 0,Y 321.875,Z 444.487,A -85,B 0,C 180,E1 -15436.099,E2 -15436.099} C_VEL
LIN {X 0,Y 320.095,Z 436.623,A -85,B 0,C 180,E1 -15439.632,E2 -15439.632} C_VEL
LIN {X 0,Y 319.592,Z 434.302,A -85,B 0,C 180,E1 -15440.798,E2 -15440.798} C_VEL
LIN {X 0,Y 318.934,Z 434.388,A -85,B 0,C 180,E1 -15441.85,E2 -15441.85} C_VEL
LIN {X 0,Y 316.101,Z 434.731,A -85,B 0,C 180,E1 -15443.562,E2 -15443.562} C_VEL
LIN {X 0,Y 313.679,Z 435.035,A -85,B 0,C 180,E1 -15444.95,E2 -15444.95} C_VEL
LIN {X 0,Y 312.616,Z 435.16,A -85,B 0,C 180,E1 -15446.024,E2 -15446.024} C_VEL
LIN {X 0,Y 312.516,Z 435.172,A -85,B 0,C 180,E1 -15446.388,E2 -15446.388} C_VEL
LIN {X 0,Y 312.551,Z 435.167,A -85,B 0,C 180,E1 -15450.35,E2 -15450.35} C_VEL
LIN {X 0,Y 312.607,Z 435.201,A -85,B 0,C 180,E1 -15451.955,E2 -15451.955} C_VEL
LIN {X 0,Y 317.245,Z 449.523,A -85,B 0,C 180,E1 -15453.36,E2 -15453.36} C_VEL
LIN {X 0,Y 321.385,Z 462.949,A -85,B 0,C 180,E1 -15454.876,E2 -15454.876} C_VEL
LIN {X 0,Y 322.398,Z 466.614,A -85,B 0,C 180,E1 -15455.323,E2 -15455.323} C_VEL
LIN {X 0,Y 320.864,Z 479.7,A -85,B 0,C 180,E1 -15456.78,E2 -15456.78} C_VEL
LIN {X 0,Y 319.136,Z 492.704,A -85,B 0,C 180,E1 -15458.524,E2 -15458.524} C_VEL
LIN {X 0,Y 317.671,Z 503.681,A -85,B 0,C 180,E1 -15460.282,E2 -15460.282} C_VEL
LIN {X 0,Y 316.207,Z 513.853,A -85,B 0,C 180,E1 -15462.205,E2 -15462.205} C_VEL
LIN {X 0,Y 315.088,Z 522.251,A -85,B 0,C 180,E1 -15464.068,E2 -15464.068} C_VEL
LIN {X 0,Y 314.082,Z 529.931,A -85,B 0,C 180,E1 -15466.081,E2 -15466.081} C_VEL
LIN {X 0,Y 313.191,Z 537.182,A -85,B 0,C 180,E1 -15468.348,E2 -15468.348} C_VEL
LIN {X 0,Y 312.455,Z 543.911,A -85,B 0,C 180,E1 -15470.941,E2 -15470.941} C_VEL
LIN {X 0,Y 311.999,Z 549.127,A -85,B 0,C 180,E1 -15473.533,E2 -15473.533} C_VEL
LIN {X 0,Y 311.912,Z 552.962,A -85,B 0,C 180,E1 -15476.124,E2 -15476.124} C_VEL
LIN {X 0,Y 311.58,Z 555.565,A -85,B 0,C 180,E1 -15478.707,E2 -15478.707} C_VEL
LIN {X 0,Y 311.609,Z 556.945,A -85,B 0,C 180,E1 -15481.292,E2 -15481.292} C_VEL
LIN {X 0,Y 312.083,Z 557.099,A -85,B 0,C 180,E1 -15483.874,E2 -15483.874} C_VEL
LIN {X 0,Y 312.882,Z 556.057,A -85,B 0,C 180,E1 -15486.448,E2 -15486.448} C_VEL
LIN {X 0,Y 313.74,Z 553.845,A -85,B 0,C 180,E1 -15489.021,E2 -15489.021} C_VEL
LIN {X 0,Y 314.963,Z 550.382,A -85,B 0,C 180,E1 -15491.585,E2 -15491.585} C_VEL
LIN {X 0,Y 316.417,Z 545.634,A -85,B 0,C 180,E1 -15494.142,E2 -15494.142} C_VEL
LIN {X 0,Y 318.471,Z 539.381,A -85,B 0,C 180,E1 -15496.671,E2 -15496.671} C_VEL
LIN {X 0,Y 320.324,Z 533.713,A -85,B 0,C 180,E1 -15498.55,E2 -15498.55} C_VEL
LIN {X 0,Y 322.753,Z 525.745,A -85,B 0,C 180,E1 -15500.723,E2 -15500.723} C_VEL
LIN {X 0,Y 325.479,Z 516.239,A -85,B 0,C 180,E1 -15502.872,E2 -15502.872} C_VEL
LIN {X 0,Y 328.665,Z 504.735,A -85,B 0,C 180,E1 -15504.981,E2 -15504.981} C_VEL
LIN {X 0,Y 331.654,Z 493.371,A -85,B 0,C 180,E1 -15506.686,E2 -15506.686} C_VEL
LIN {X 0,Y 334.747,Z 479.83,A -85,B 0,C 180,E1 -15508.404,E2 -15508.404} C_VEL
LIN {X 0,Y 334.324,Z 476.974,A -85,B 0,C 180,E1 -15508.914,E2 -15508.914} C_VEL
LIN {X 0,Y 331.718,Z 468.169,A -85,B 0,C 180,E1 -15510.78,E2 -15510.78} C_VEL
LIN {X 0,Y 327.931,Z 459.193,A -85,B 0,C 180,E1 -15513.062,E2 -15513.062} C_VEL
LIN {X 0,Y 324.195,Z 452.539,A -85,B 0,C 180,E1 -15515.216,E2 -15515.216} C_VEL
LIN {X 0,Y 322.388,Z 450.561,A -85,B 0,C 180,E1 -15516.236,E2 -15516.236} C_VEL
LIN {X 0,Y 319.324,Z 448.352,A -85,B 0,C 180,E1 -15518.043,E2 -15518.043} C_VEL
LIN {X 0,Y 317.773,Z 446.819,A -85,B 0,C 180,E1 -15519.279,E2 -15519.279} C_VEL
LIN {X 0,Y 315.796,Z 446.898,A -85,B 0,C 180,E1 -15520.829,E2 -15520.829} C_VEL
LIN {X 0,Y 314.271,Z 446.522,A -85,B 0,C 180,E1 -15523.373,E2 -15523.373} C_VEL
LIN {X 0,Y 313.725,Z 450.229,A -85,B 0,C 180,E1 -15526.016,E2 -15526.016} C_VEL
LIN {X 0,Y 313.41,Z 453.012,A -85,B 0,C 180,E1 -15527.731,E2 -15527.731} C_VEL
LIN {X 0,Y 314.437,Z 460.638,A -85,B 0,C 180,E1 -15530.454,E2 -15530.454} C_VEL
LIN {X 0,Y 316.423,Z 466.064,A -85,B 0,C 180,E1 -15532.377,E2 -15532.377} C_VEL
LIN {X 0,Y 317.444,Z 471.032,A -85,B 0,C 180,E1 -15533.507,E2 -15533.507} C_VEL
LIN {X 0,Y 318.385,Z 473.666,A -85,B 0,C 180,E1 -15534.206,E2 -15534.206} C_VEL
LIN {X 0,Y 319.934,Z 479.939,A -85,B 0,C 180,E1 -15535.483,E2 -15535.483} C_VEL
LIN {X 0,Y 320.697,Z 482.549,A -85,B 0,C 180,E1 -15536.025,E2 -15536.025} C_VEL
LIN {X 0,Y 323.329,Z 495.236,A -85,B 0,C 180,E1 -15538.177,E2 -15538.177} C_VEL
LIN {X 0,Y 324.956,Z 506.944,A -85,B 0,C 180,E1 -15539.894,E2 -15539.894} C_VEL
LIN {X 0,Y 325.558,Z 518.863,A -85,B 0,C 180,E1 -15541.476,E2 -15541.476} C_VEL
LIN {X 0,Y 325.224,Z 528.408,A -85,B 0,C 180,E1 -15542.689,E2 -15542.689} C_VEL
LIN {X 0,Y 323.992,Z 543,A -85,B 0,C 180,E1 -15544.633,E2 -15544.633} C_VEL
LIN {X 0,Y 323.587,Z 549.639,A -85,B 0,C 180,E1 -15545.628,E2 -15545.628} C_VEL
LIN {X 0,Y 322.609,Z 553.642,A -85,B 0,C 180,E1 -15546.158,E2 -15546.158} C_VEL
LIN {X 0,Y 320.911,Z 565.827,A -85,B 0,C 180,E1 -15547.465,E2 -15547.465} C_VEL
LIN {X 0,Y 318.94,Z 577.549,A -85,B 0,C 180,E1 -15549.018,E2 -15549.018} C_VEL
LIN {X 0,Y 317.233,Z 587.238,A -85,B 0,C 180,E1 -15550.591,E2 -15550.591} C_VEL
LIN {X 0,Y 315.48,Z 596.911,A -85,B 0,C 180,E1 -15552.498,E2 -15552.498} C_VEL
LIN {X 0,Y 314.158,Z 604.915,A -85,B 0,C 180,E1 -15554.428,E2 -15554.428} C_VEL
LIN {X 0,Y 313.024,Z 611.564,A -85,B 0,C 180,E1 -15556.364,E2 -15556.364} C_VEL
LIN {X 0,Y 312.026,Z 617.074,A -85,B 0,C 180,E1 -15558.304,E2 -15558.304} C_VEL
LIN {X 0,Y 311.291,Z 622.836,A -85,B 0,C 180,E1 -15560.907,E2 -15560.907} C_VEL
LIN {X 0,Y 310.9,Z 627.016,A -85,B 0,C 180,E1 -15563.51,E2 -15563.51} C_VEL
LIN {X 0,Y 310.757,Z 629.747,A -85,B 0,C 180,E1 -15566.11,E2 -15566.11} C_VEL
LIN {X 0,Y 310.681,Z 631.102,A -85,B 0,C 180,E1 -15568.704,E2 -15568.704} C_VEL
LIN {X 0,Y 310.681,Z 631.099,A -85,B 0,C 180,E1 -15571.296,E2 -15571.296} C_VEL
LIN {X 0,Y 310.75,Z 629.74,A -85,B 0,C 180,E1 -15573.89,E2 -15573.89} C_VEL
LIN {X 0,Y 310.888,Z 627.005,A -85,B 0,C 180,E1 -15576.49,E2 -15576.49} C_VEL
LIN {X 0,Y 311.28,Z 622.814,A -85,B 0,C 180,E1 -15579.093,E2 -15579.093} C_VEL
LIN {X 0,Y 312.019,Z 617.043,A -85,B 0,C 180,E1 -15581.696,E2 -15581.696} C_VEL
LIN {X 0,Y 313.181,Z 610.521,A -85,B 0,C 180,E1 -15583.96,E2 -15583.96} C_VEL
LIN {X 0,Y 314.434,Z 602.595,A -85,B 0,C 180,E1 -15586.172,E2 -15586.172} C_VEL
LIN {X 0,Y 316.008,Z 593.867,A -85,B 0,C 180,E1 -15588.141,E2 -15588.141} C_VEL
LIN {X 0,Y 317.831,Z 583.504,A -85,B 0,C 180,E1 -15590.044,E2 -15590.044} C_VEL
LIN {X 0,Y 319.662,Z 573.061,A -85,B 0,C 180,E1 -15591.608,E2 -15591.608} C_VEL
LIN {X 0,Y 321.49,Z 561.674,A -85,B 0,C 180,E1 -15593.002,E2 -15593.002} C_VEL
LIN {X 0,Y 323.028,Z 550.354,A -85,B 0,C 180,E1 -15594.131,E2 -15594.131} C_VEL
LIN {X 0,Y 323.069,Z 546.136,A -85,B 0,C 180,E1 -15594.536,E2 -15594.536} C_VEL
LIN {X 0,Y 321.818,Z 533.093,A -85,B 0,C 180,E1 -15595.701,E2 -15595.701} C_VEL
LIN {X 0,Y 319.7,Z 519.109,A -85,B 0,C 180,E1 -15596.736,E2 -15596.736} C_VEL
LIN {X 0,Y 317.013,Z 504.521,A -85,B 0,C 180,E1 -15597.578,E2 -15597.578} C_VEL
LIN {X 0,Y 314.674,Z 494.844,A -85,B 0,C 180,E1 -15598.063,E2 -15598.063} C_VEL
LIN {X 0,Y 313.06,Z 489.426,A -85,B 0,C 180,E1 -15598.402,E2 -15598.402} C_VEL
LIN {X 0,Y 312.477,Z 484.043,A -85,B 0,C 180,E1 -15599.238,E2 -15599.238} C_VEL
LIN {X 0,Y 313.087,Z 476.963,A -85,B 0,C 180,E1 -15603.241,E2 -15603.241} C_VEL
LIN {X 0,Y 313.462,Z 471.867,A -85,B 0,C 180,E1 -15606.182,E2 -15606.182} C_VEL
LIN {X 0,Y 314.026,Z 465.936,A -85,B 0,C 180,E1 -15609.631,E2 -15609.631} C_VEL
LIN {X 0,Y 314.753,Z 458.987,A -85,B 0,C 180,E1 -15613.804,E2 -15613.804} C_VEL
LIN {X 0,Y 315.297,Z 453.212,A -85,B 0,C 180,E1 -15617.356,E2 -15617.356} C_VEL
LIN {X 0,Y 315.053,Z 449.609,A -85,B 0,C 180,E1 -15619.691,E2 -15619.691} C_VEL
LIN {X 0,Y 314.038,Z 443.75,A -85,B 0,C 180,E1 -15623.674,E2 -15623.674} C_VEL
LIN {X 0,Y 313.156,Z 438.506,A -85,B 0,C 180,E1 -15627.41,E2 -15627.41} C_VEL
LIN {X 0,Y 312.585,Z 435.177,A -85,B 0,C 180,E1 -15629.983,E2 -15629.983} C_VEL
LIN {X 0,Y 312.604,Z 435.153,A -85,B 0,C 180,E1 -15634.064,E2 -15634.064} C_VEL
LIN {X 0,Y 312.589,Z 435.169,A -85,B 0,C 180,E1 -15637.529,E2 -15637.529} C_VEL
LIN {X 0,Y 312.64,Z 435.165,A -85,B 0,C 180,E1 -15641.657,E2 -15641.657} C_VEL
LIN {X 0,Y 312.695,Z 435.141,A -85,B 0,C 180,E1 -15645.686,E2 -15645.686} C_VEL
LIN {X 0,Y 312.687,Z 435.152,A -85,B 0,C 180,E1 -15649.641,E2 -15649.641} C_VEL
LIN {X 0,Y 312.895,Z 435.134,A -85,B 0,C 180,E1 -15653.552,E2 -15653.552} C_VEL
LIN {X 0,Y 312.938,Z 435.11,A -85,B 0,C 180,E1 -15657.426,E2 -15657.426} C_VEL
LIN {X 0,Y 313.122,Z 435.109,A -85,B 0,C 180,E1 -15660,E2 -15660} C_VEL
LIN {X 0,Y 312.937,Z 435.111,A -85,B 0,C 180,E1 -15662.574,E2 -15662.574} C_VEL
LIN {X 0,Y 312.896,Z 435.13,A -85,B 0,C 180,E1 -15666.639,E2 -15666.639} C_VEL
LIN {X 0,Y 312.789,Z 435.131,A -85,B 0,C 180,E1 -15669.049,E2 -15669.049} C_VEL
LIN {X 0,Y 312.636,Z 435.156,A -85,B 0,C 180,E1 -15672.991,E2 -15672.991} C_VEL
LIN {X 0,Y 312.64,Z 435.167,A -85,B 0,C 180,E1 -15675.65,E2 -15675.65} C_VEL
LIN {X 0,Y 312.61,Z 435.159,A -85,B 0,C 180,E1 -15679.225,E2 -15679.225} C_VEL
LIN {X 0,Y 312.527,Z 435.17,A -85,B 0,C 180,E1 -15682.781,E2 -15682.781} C_VEL
LIN {X 0,Y 312.604,Z 435.165,A -85,B 0,C 180,E1 -15685.936,E2 -15685.936} C_VEL
LIN {X 0,Y 312.547,Z 435.173,A -85,B 0,C 180,E1 -15689.65,E2 -15689.65} C_VEL
LIN {X 0,Y 312.521,Z 435.178,A -85,B 0,C 180,E1 -15693.689,E2 -15693.689} C_VEL
LIN {X 0,Y 312.527,Z 435.179,A -85,B 0,C 180,E1 -15697.385,E2 -15697.385} C_VEL
LIN {X 0,Y 312.572,Z 435.373,A -85,B 0,C 180,E1 -15698.729,E2 -15698.729} C_VEL
LIN {X 0,Y 314.427,Z 443.373,A -85,B 0,C 180,E1 -15702.472,E2 -15702.472} C_VEL
LIN {X 0,Y 315.995,Z 451.058,A -85,B 0,C 180,E1 -15705.933,E2 -15705.933} C_VEL
LIN {X 0,Y 317.127,Z 457.771,A -85,B 0,C 180,E1 -15708.894,E2 -15708.894} C_VEL
LIN {X 0,Y 317.232,Z 461.769,A -85,B 0,C 180,E1 -15710.539,E2 -15710.539} C_VEL
LIN {X 0,Y 316.301,Z 472.39,A -85,B 0,C 180,E1 -15714.711,E2 -15714.711} C_VEL
LIN {X 0,Y 315.594,Z 482.267,A -85,B 0,C 180,E1 -15718.475,E2 -15718.475} C_VEL
LIN {X 0,Y 315.001,Z 491.478,A -85,B 0,C 180,E1 -15721.788,E2 -15721.788} C_VEL
LIN {X 0,Y 319.562,Z 507.513,A -85,B 0,C 180,E1 -15722.745,E2 -15722.745} C_VEL
LIN {X 0,Y 322.487,Z 521.167,A -85,B 0,C 180,E1 -15723.723,E2 -15723.723} C_VEL
LIN {X 0,Y 324.494,Z 534.962,A -85,B 0,C 180,E1 -15724.888,E2 -15724.888} C_VEL
LIN {X 0,Y 324.44,Z 538.684,A -85,B 0,C 180,E1 -15725.209,E2 -15725.209} C_VEL
LIN {X 0,Y 323.04,Z 550.513,A -85,B 0,C 180,E1 -15726.274,E2 -15726.274} C_VEL
LIN {X 0,Y 321.202,Z 562.87,A -85,B 0,C 180,E1 -15727.656,E2 -15727.656} C_VEL
LIN {X 0,Y 319.18,Z 574.12,A -85,B 0,C 180,E1 -15729.203,E2 -15729.203} C_VEL
LIN {X 0,Y 317.366,Z 584.334,A -85,B 0,C 180,E1 -15730.935,E2 -15730.935} C_VEL
LIN {X 0,Y 315.572,Z 593.562,A -85,B 0,C 180,E1 -15732.837,E2 -15732.837} C_VEL
LIN {X 0,Y 314.296,Z 601.216,A -85,B 0,C 180,E1 -15734.767,E2 -15734.767} C_VEL
LIN {X 0,Y 312.899,Z 608.536,A -85,B 0,C 180,E1 -15737.02,E2 -15737.02} C_VEL
LIN {X 0,Y 311.827,Z 615.082,A -85,B 0,C 180,E1 -15739.612,E2 -15739.612} C_VEL
LIN {X 0,Y 311.165,Z 619.994,A -85,B 0,C 180,E1 -15742.212,E2 -15742.212} C_VEL
LIN {X 0,Y 310.801,Z 623.415,A -85,B 0,C 180,E1 -15744.81,E2 -15744.81} C_VEL
LIN {X 0,Y 310.679,Z 625.447,A -85,B 0,C 180,E1 -15747.407,E2 -15747.407} C_VEL
LIN {X 0,Y 310.617,Z 626.145,A -85,B 0,C 180,E1 -15750,E2 -15750} C_VEL
LIN {X 0,Y 310.679,Z 625.509,A -85,B 0,C 180,E1 -15752.593,E2 -15752.593} C_VEL
LIN {X 0,Y 310.781,Z 623.528,A -85,B 0,C 180,E1 -15755.19,E2 -15755.19} C_VEL
LIN {X 0,Y 311.164,Z 620.162,A -85,B 0,C 180,E1 -15757.789,E2 -15757.789} C_VEL
LIN {X 0,Y 311.808,Z 615.312,A -85,B 0,C 180,E1 -15760.388,E2 -15760.388} C_VEL
LIN {X 0,Y 312.865,Z 608.826,A -85,B 0,C 180,E1 -15762.981,E2 -15762.981} C_VEL
LIN {X 0,Y 314.225,Z 601.591,A -85,B 0,C 180,E1 -15765.236,E2 -15765.236} C_VEL
LIN {X 0,Y 315.6,Z 594,A -85,B 0,C 180,E1 -15767.161,E2 -15767.161} C_VEL
LIN {X 0,Y 317.305,Z 584.881,A -85,B 0,C 180,E1 -15769.068,E2 -15769.068} C_VEL
LIN {X 0,Y 319.103,Z 574.792,A -85,B 0,C 180,E1 -15770.802,E2 -15770.802} C_VEL
LIN {X 0,Y 321.059,Z 563.678,A -85,B 0,C 180,E1 -15772.355,E2 -15772.355} C_VEL
LIN {X 0,Y 322.84,Z 552.104,A -85,B 0,C 180,E1 -15773.674,E2 -15773.674} C_VEL
LIN {X 0,Y 324.439,Z 539.633,A -85,B 0,C 180,E1 -15774.816,E2 -15774.816} C_VEL
LIN {X 0,Y 324.526,Z 534.734,A -85,B 0,C 180,E1 -15775.237,E2 -15775.237} C_VEL
LIN {X 0,Y 322.558,Z 521.381,A -85,B 0,C 180,E1 -15776.369,E2 -15776.369} C_VEL
LIN {X 0,Y 319.496,Z 507.198,A -85,B 0,C 180,E1 -15777.386,E2 -15777.386} C_VEL
LIN {X 0,Y 314.987,Z 491.256,A -85,B 0,C 180,E1 -15778.355,E2 -15778.355} C_VEL
LIN {X 0,Y 315.569,Z 482.616,A -85,B 0,C 180,E1 -15781.519,E2 -15781.519} C_VEL
LIN {X 0,Y 316.308,Z 472.69,A -85,B 0,C 180,E1 -15785.288,E2 -15785.288} C_VEL
LIN {X 0,Y 317.227,Z 462.067,A -85,B 0,C 180,E1 -15789.461,E2 -15789.461} C_VEL
LIN {X 0,Y 317.179,Z 458.075,A -85,B 0,C 180,E1 -15791.117,E2 -15791.117} C_VEL
LIN {X 0,Y 316.1,Z 451.345,A -85,B 0,C 180,E1 -15794.072,E2 -15794.072} C_VEL
LIN {X 0,Y 314.359,Z 442.987,A -85,B 0,C 180,E1 -15797.879,E2 -15797.879} C_VEL
LIN {X 0,Y 312.551,Z 435.183,A -85,B 0,C 180,E1 -15801.502,E2 -15801.502} C_VEL
LIN {X 0,Y 312.534,Z 435.181,A -85,B 0,C 180,E1 -15804.22,E2 -15804.22} C_VEL
LIN {X 0,Y 312.516,Z 435.172,A -85,B 0,C 180,E1 -15806.388,E2 -15806.388} C_VEL
LIN {X 0,Y 311.814,Z 435.267,A -85,B 0,C 180,E1 -15807.104,E2 -15807.104} C_VEL
LIN {X 0,Y 308.964,Z 435.623,A -85,B 0,C 180,E1 -15808.226,E2 -15808.226} C_VEL
LIN {X 0,Y 306.123,Z 435.967,A -85,B 0,C 180,E1 -15809.368,E2 -15809.368} C_VEL
LIN {X 0,Y 305.461,Z 436.048,A -85,B 0,C 180,E1 -15810.107,E2 -15810.107} C_VEL
LIN {X 0,Y 305.535,Z 436.053,A -85,B 0,C 180,E1 -15811.527,E2 -15811.527} C_VEL
LIN {X 0,Y 310.179,Z 450.2,A -85,B 0,C 180,E1 -15812.953,E2 -15812.953} C_VEL
LIN {X 0,Y 314.611,Z 464.802,A -85,B 0,C 180,E1 -15814.651,E2 -15814.651} C_VEL
LIN {X 0,Y 315.421,Z 468.674,A -85,B 0,C 180,E1 -15815.13,E2 -15815.13} C_VEL
LIN {X 0,Y 313.703,Z 482.319,A -85,B 0,C 180,E1 -15816.713,E2 -15816.713} C_VEL
LIN {X 0,Y 311.992,Z 495.227,A -85,B 0,C 180,E1 -15818.528,E2 -15818.528} C_VEL
LIN {X 0,Y 310.384,Z 506.853,A -85,B 0,C 180,E1 -15820.489,E2 -15820.489} C_VEL
LIN {X 0,Y 308.68,Z 518.19,A -85,B 0,C 180,E1 -15822.783,E2 -15822.783} C_VEL
LIN {X 0,Y 307.571,Z 527.586,A -85,B 0,C 180,E1 -15825.104,E2 -15825.104} C_VEL
LIN {X 0,Y 306.448,Z 535.391,A -85,B 0,C 180,E1 -15827.416,E2 -15827.416} C_VEL
LIN {X 0,Y 305.632,Z 542.636,A -85,B 0,C 180,E1 -15830.069,E2 -15830.069} C_VEL
LIN {X 0,Y 305.126,Z 547.805,A -85,B 0,C 180,E1 -15832.431,E2 -15832.431} C_VEL
LIN {X 0,Y 304.922,Z 551.684,A -85,B 0,C 180,E1 -15834.71,E2 -15834.71} C_VEL
LIN {X 0,Y 304.853,Z 553.51,A -85,B 0,C 180,E1 -15836.034,E2 -15836.034} C_VEL
LIN {X 0,Y 304.539,Z 556.242,A -85,B 0,C 180,E1 -15838.678,E2 -15838.678} C_VEL
LIN {X 0,Y 304.567,Z 557.745,A -85,B 0,C 180,E1 -15841.322,E2 -15841.322} C_VEL
LIN {X 0,Y 305.064,Z 558.03,A -85,B 0,C 180,E1 -15843.963,E2 -15843.963} C_VEL
LIN {X 0,Y 305.904,Z 557.112,A -85,B 0,C 180,E1 -15846.596,E2 -15846.596} C_VEL
LIN {X 0,Y 306.832,Z 555.038,A -85,B 0,C 180,E1 -15849.226,E2 -15849.226} C_VEL
LIN {X 0,Y 308.149,Z 551.73,A -85,B 0,C 180,E1 -15851.845,E2 -15851.845} C_VEL
LIN {X 0,Y 309.705,Z 547.125,A -85,B 0,C 180,E1 -15854.455,E2 -15854.455} C_VEL
LIN {X 0,Y 311.875,Z 541.087,A -85,B 0,C 180,E1 -15857.035,E2 -15857.035} C_VEL
LIN {X 0,Y 314.196,Z 534.506,A -85,B 0,C 180,E1 -15859.265,E2 -15859.265} C_VEL
LIN {X 0,Y 316.819,Z 526.614,A -85,B 0,C 180,E1 -15861.47,E2 -15861.47} C_VEL
LIN {X 0,Y 320.203,Z 515.631,A -85,B 0,C 180,E1 -15863.957,E2 -15863.957} C_VEL
LIN {X 0,Y 323.162,Z 505.702,A -85,B 0,C 180,E1 -15865.782,E2 -15865.782} C_VEL
LIN {X 0,Y 326.233,Z 494.998,A -85,B 0,C 180,E1 -15867.435,E2 -15867.435} C_VEL
LIN {X 0,Y 329.256,Z 482.889,A -85,B 0,C 180,E1 -15869.017,E2 -15869.017} C_VEL
LIN {X 0,Y 328.827,Z 479.667,A -85,B 0,C 180,E1 -15869.658,E2 -15869.658} C_VEL
LIN {X 0,Y 326.711,Z 471.886,A -85,B 0,C 180,E1 -15871.443,E2 -15871.443} C_VEL
LIN {X 0,Y 323.754,Z 464.497,A -85,B 0,C 180,E1 -15873.454,E2 -15873.454} C_VEL
LIN {X 0,Y 321.273,Z 459.516,A -85,B 0,C 180,E1 -15875.136,E2 -15875.136} C_VEL
LIN {X 0,Y 320.39,Z 458.081,A -85,B 0,C 180,E1 -15875.745,E2 -15875.745} C_VEL
LIN {X 0,Y 319.165,Z 456.795,A -85,B 0,C 180,E1 -15876.48,E2 -15876.48} C_VEL
LIN {X 0,Y 315.799,Z 454.053,A -85,B 0,C 180,E1 -15878.839,E2 -15878.839} C_VEL
LIN {X 0,Y 313.738,Z 453.581,A -85,B 0,C 180,E1 -15880.513,E2 -15880.513} C_VEL
LIN {X 0,Y 312.366,Z 453.271,A -85,B 0,C 180,E1 -15882.452,E2 -15882.452} C_VEL
LIN {X 0,Y 311.63,Z 453.903,A -85,B 0,C 180,E1 -15883.807,E2 -15883.807} C_VEL
LIN {X 0,Y 310.867,Z 457.525,A -85,B 0,C 180,E1 -15886.34,E2 -15886.34} C_VEL
LIN {X 0,Y 310.933,Z 459.252,A -85,B 0,C 180,E1 -15887.305,E2 -15887.305} C_VEL
LIN {X 0,Y 311.581,Z 466.821,A -85,B 0,C 180,E1 -15890.076,E2 -15890.076} C_VEL
LIN {X 0,Y 313.033,Z 471.506,A -85,B 0,C 180,E1 -15891.794,E2 -15891.794} C_VEL
LIN {X 0,Y 313.967,Z 476.81,A -85,B 0,C 180,E1 -15893.084,E2 -15893.084} C_VEL
LIN {X 0,Y 314.781,Z 479.645,A -85,B 0,C 180,E1 -15893.835,E2 -15893.835} C_VEL
LIN {X 0,Y 315.802,Z 484.843,A -85,B 0,C 180,E1 -15894.934,E2 -15894.934} C_VEL
LIN {X 0,Y 316.294,Z 486.398,A -85,B 0,C 180,E1 -15895.299,E2 -15895.299} C_VEL
LIN {X 0,Y 318.383,Z 499.019,A -85,B 0,C 180,E1 -15897.574,E2 -15897.574} C_VEL
LIN {X 0,Y 319.592,Z 510.565,A -85,B 0,C 180,E1 -15899.367,E2 -15899.367} C_VEL
LIN {X 0,Y 319.766,Z 522.701,A -85,B 0,C 180,E1 -15901.084,E2 -15901.084} C_VEL
LIN {X 0,Y 318.804,Z 534.036,A -85,B 0,C 180,E1 -15902.601,E2 -15902.601} C_VEL
LIN {X 0,Y 317.47,Z 547.617,A -85,B 0,C 180,E1 -15904.601,E2 -15904.601} C_VEL
LIN {X 0,Y 317.221,Z 550.79,A -85,B 0,C 180,E1 -15905.106,E2 -15905.106} C_VEL
LIN {X 0,Y 315.672,Z 556.568,A -85,B 0,C 180,E1 -15905.93,E2 -15905.93} C_VEL
LIN {X 0,Y 313.954,Z 568.358,A -85,B 0,C 180,E1 -15907.285,E2 -15907.285} C_VEL
LIN {X 0,Y 311.876,Z 579.629,A -85,B 0,C 180,E1 -15908.866,E2 -15908.866} C_VEL
LIN {X 0,Y 309.892,Z 590.635,A -85,B 0,C 180,E1 -15910.801,E2 -15910.801} C_VEL
LIN {X 0,Y 308.165,Z 599.696,A -85,B 0,C 180,E1 -15912.754,E2 -15912.754} C_VEL
LIN {X 0,Y 306.608,Z 608.339,A -85,B 0,C 180,E1 -15915.056,E2 -15915.056} C_VEL
LIN {X 0,Y 305.358,Z 615.298,A -85,B 0,C 180,E1 -15917.37,E2 -15917.37} C_VEL
LIN {X 0,Y 304.408,Z 621.526,A -85,B 0,C 180,E1 -15920.029,E2 -15920.029} C_VEL
LIN {X 0,Y 304.004,Z 625.057,A -85,B 0,C 180,E1 -15922.027,E2 -15922.027} C_VEL
LIN {X 0,Y 303.693,Z 628.499,A -85,B 0,C 180,E1 -15924.689,E2 -15924.689} C_VEL
LIN {X 0,Y 303.647,Z 630.536,A -85,B 0,C 180,E1 -15927.347,E2 -15927.347} C_VEL
LIN {X 0,Y 303.591,Z 631.211,A -85,B 0,C 180,E1 -15930,E2 -15930} C_VEL
LIN {X 0,Y 303.646,Z 630.53,A -85,B 0,C 180,E1 -15932.653,E2 -15932.653} C_VEL
LIN {X 0,Y 303.685,Z 628.489,A -85,B 0,C 180,E1 -15935.311,E2 -15935.311} C_VEL
LIN {X 0,Y 303.986,Z 625.039,A -85,B 0,C 180,E1 -15937.974,E2 -15937.974} C_VEL
LIN {X 0,Y 304.59,Z 620.076,A -85,B 0,C 180,E1 -15940.637,E2 -15940.637} C_VEL
LIN {X 0,Y 305.35,Z 615.261,A -85,B 0,C 180,E1 -15942.63,E2 -15942.63} C_VEL
LIN {X 0,Y 306.551,Z 608.294,A -85,B 0,C 180,E1 -15944.947,E2 -15944.947} C_VEL
LIN {X 0,Y 308.112,Z 599.639,A -85,B 0,C 180,E1 -15947.249,E2 -15947.249} C_VEL
LIN {X 0,Y 309.817,Z 590.567,A -85,B 0,C 180,E1 -15949.203,E2 -15949.203} C_VEL
LIN {X 0,Y 311.848,Z 579.539,A -85,B 0,C 180,E1 -15951.136,E2 -15951.136} C_VEL
LIN {X 0,Y 313.88,Z 568.247,A -85,B 0,C 180,E1 -15952.721,E2 -15952.721} C_VEL
LIN {X 0,Y 315.699,Z 556.01,A -85,B 0,C 180,E1 -15954.115,E2 -15954.115} C_VEL
LIN {X 0,Y 316.597,Z 548.939,A -85,B 0,C 180,E1 -15954.79,E2 -15954.79} C_VEL
LIN {X 0,Y 315.558,Z 536.46,A -85,B 0,C 180,E1 -15955.986,E2 -15955.986} C_VEL
LIN {X 0,Y 313.61,Z 522.334,A -85,B 0,C 180,E1 -15957.122,E2 -15957.122} C_VEL
LIN {X 0,Y 311.085,Z 507.649,A -85,B 0,C 180,E1 -15958.051,E2 -15958.051} C_VEL
LIN {X 0,Y 308.926,Z 498.045,A -85,B 0,C 180,E1 -15958.552,E2 -15958.552} C_VEL
LIN {X 0,Y 306.333,Z 489.56,A -85,B 0,C 180,E1 -15959.075,E2 -15959.075} C_VEL
LIN {X 0,Y 305.542,Z 482.606,A -85,B 0,C 180,E1 -15960.215,E2 -15960.215} C_VEL
LIN {X 0,Y 306.175,Z 475.62,A -85,B 0,C 180,E1 -15964.274,E2 -15964.274} C_VEL
LIN {X 0,Y 306.825,Z 467.891,A -85,B 0,C 180,E1 -15968.85,E2 -15968.85} C_VEL
LIN {X 0,Y 307.599,Z 460.64,A -85,B 0,C 180,E1 -15973.27,E2 -15973.27} C_VEL
LIN {X 0,Y 308.183,Z 454.894,A -85,B 0,C 180,E1 -15976.865,E2 -15976.865} C_VEL
LIN {X 0,Y 308.07,Z 450.8,A -85,B 0,C 180,E1 -15979.553,E2 -15979.553} C_VEL
LIN {X 0,Y 307.059,Z 445.11,A -85,B 0,C 180,E1 -15983.481,E2 -15983.481} C_VEL
LIN {X 0,Y 306.179,Z 439.736,A -85,B 0,C 180,E1 -15987.356,E2 -15987.356} C_VEL
LIN {X 0,Y 305.548,Z 436.054,A -85,B 0,C 180,E1 -15990.248,E2 -15990.248} C_VEL
LIN {X 0,Y 305.572,Z 436.029,A -85,B 0,C 180,E1 -15994.088,E2 -15994.088} C_VEL
LIN {X 0,Y 305.502,Z 436.042,A -85,B 0,C 180,E1 -15998.403,E2 -15998.403} C_VEL
LIN {X 0,Y 305.592,Z 436.041,A -85,B 0,C 180,E1 -16001.218,E2 -16001.218} C_VEL
LIN {X 0,Y 305.65,Z 436.017,A -85,B 0,C 180,E1 -16005.349,E2 -16005.349} C_VEL
LIN {X 0,Y 305.626,Z 436.033,A -85,B 0,C 180,E1 -16009.399,E2 -16009.399} C_VEL
LIN {X 0,Y 305.773,Z 436.006,A -85,B 0,C 180,E1 -16012.073,E2 -16012.073} C_VEL
LIN {X 0,Y 305.687,Z 436.032,A -85,B 0,C 180,E1 -16014.724,E2 -16014.724} C_VEL
LIN {X 0,Y 305.959,Z 435.99,A -85,B 0,C 180,E1 -16018.684,E2 -16018.684} C_VEL
LIN {X 0,Y 305.959,Z 435.992,A -85,B 0,C 180,E1 -16021.316,E2 -16021.316} C_VEL
LIN {X 0,Y 305.852,Z 436.01,A -85,B 0,C 180,E1 -16026.617,E2 -16026.617} C_VEL
LIN {X 0,Y 305.737,Z 436.01,A -85,B 0,C 180,E1 -16029.26,E2 -16029.26} C_VEL
LIN {X 0,Y 305.59,Z 436.031,A -85,B 0,C 180,E1 -16033.296,E2 -16033.296} C_VEL
LIN {X 0,Y 305.596,Z 436.045,A -85,B 0,C 180,E1 -16036.02,E2 -16036.02} C_VEL
LIN {X 0,Y 305.562,Z 436.039,A -85,B 0,C 180,E1 -16039.436,E2 -16039.436} C_VEL
LIN {X 0,Y 305.487,Z 436.046,A -85,B 0,C 180,E1 -16043.039,E2 -16043.039} C_VEL
LIN {X 0,Y 305.549,Z 436.042,A -85,B 0,C 180,E1 -16046.227,E2 -16046.227} C_VEL
LIN {X 0,Y 305.497,Z 436.055,A -85,B 0,C 180,E1 -16049.05,E2 -16049.05} C_VEL
LIN {X 0,Y 305.446,Z 436.064,A -85,B 0,C 180,E1 -16051.952,E2 -16051.952} C_VEL
LIN {X 0,Y 305.464,Z 436.057,A -85,B 0,C 180,E1 -16055.113,E2 -16055.113} C_VEL
LIN {X 0,Y 305.504,Z 436.257,A -85,B 0,C 180,E1 -16057.875,E2 -16057.875} C_VEL
LIN {X 0,Y 307.312,Z 443.837,A -85,B 0,C 180,E1 -16061.545,E2 -16061.545} C_VEL
LIN {X 0,Y 308.972,Z 451.666,A -85,B 0,C 180,E1 -16065.159,E2 -16065.159} C_VEL
LIN {X 0,Y 310.223,Z 458.788,A -85,B 0,C 180,E1 -16068.384,E2 -16068.384} C_VEL
LIN {X 0,Y 310.428,Z 463.417,A -85,B 0,C 180,E1 -16070.332,E2 -16070.332} C_VEL
LIN {X 0,Y 309.49,Z 473.75,A -85,B 0,C 180,E1 -16074.441,E2 -16074.441} C_VEL
LIN {X 0,Y 308.704,Z 484.079,A -85,B 0,C 180,E1 -16078.425,E2 -16078.425} C_VEL
LIN {X 0,Y 308.177,Z 491.348,A -85,B 0,C 180,E1 -16081.104,E2 -16081.104} C_VEL
LIN {X 0,Y 312.825,Z 507.534,A -85,B 0,C 180,E1 -16082.108,E2 -16082.108} C_VEL
LIN {X 0,Y 315.818,Z 521.245,A -85,B 0,C 180,E1 -16083.127,E2 -16083.127} C_VEL
LIN {X 0,Y 317.66,Z 533.481,A -85,B 0,C 180,E1 -16084.187,E2 -16084.187} C_VEL
LIN {X 0,Y 317.973,Z 538.969,A -85,B 0,C 180,E1 -16084.692,E2 -16084.692} C_VEL
LIN {X 0,Y 316.463,Z 551.147,A -85,B 0,C 180,E1 -16085.817,E2 -16085.817} C_VEL
LIN {X 0,Y 314.624,Z 562.92,A -85,B 0,C 180,E1 -16087.162,E2 -16087.162} C_VEL
LIN {X 0,Y 312.511,Z 574.173,A -85,B 0,C 180,E1 -16088.738,E2 -16088.738} C_VEL
LIN {X 0,Y 310.649,Z 584.389,A -85,B 0,C 180,E1 -16090.507,E2 -16090.507} C_VEL
LIN {X 0,Y 308.758,Z 593.618,A -85,B 0,C 180,E1 -16092.446,E2 -16092.446} C_VEL
LIN {X 0,Y 307.389,Z 601.273,A -85,B 0,C 180,E1 -16094.416,E2 -16094.416} C_VEL
LIN {X 0,Y 305.978,Z 608.594,A -85,B 0,C 180,E1 -16096.721,E2 -16096.721} C_VEL
LIN {X 0,Y 304.805,Z 615.141,A -85,B 0,C 180,E1 -16099.37,E2 -16099.37} C_VEL
LIN {X 0,Y 304.098,Z 620.053,A -85,B 0,C 180,E1 -16102.029,E2 -16102.029} C_VEL
LIN {X 0,Y 303.717,Z 623.474,A -85,B 0,C 180,E1 -16104.689,E2 -16104.689} C_VEL
LIN {X 0,Y 303.606,Z 625.506,A -85,B 0,C 180,E1 -16107.346,E2 -16107.346} C_VEL
LIN {X 0,Y 303.533,Z 626.203,A -85,B 0,C 180,E1 -16110,E2 -16110} C_VEL
LIN {X 0,Y 303.605,Z 625.567,A -85,B 0,C 180,E1 -16112.654,E2 -16112.654} C_VEL
LIN {X 0,Y 303.691,Z 623.586,A -85,B 0,C 180,E1 -16115.311,E2 -16115.311} C_VEL
LIN {X 0,Y 304.097,Z 620.219,A -85,B 0,C 180,E1 -16117.971,E2 -16117.971} C_VEL
LIN {X 0,Y 304.781,Z 615.369,A -85,B 0,C 180,E1 -16120.63,E2 -16120.63} C_VEL
LIN {X 0,Y 305.572,Z 610.666,A -85,B 0,C 180,E1 -16122.621,E2 -16122.621} C_VEL
LIN {X 0,Y 307.002,Z 603.847,A -85,B 0,C 180,E1 -16124.924,E2 -16124.924} C_VEL
LIN {X 0,Y 308.509,Z 595.386,A -85,B 0,C 180,E1 -16127.226,E2 -16127.226} C_VEL
LIN {X 0,Y 310.251,Z 586.536,A -85,B 0,C 180,E1 -16129.176,E2 -16129.176} C_VEL
LIN {X 0,Y 312.255,Z 575.823,A -85,B 0,C 180,E1 -16131.107,E2 -16131.107} C_VEL
LIN {X 0,Y 314.282,Z 564.952,A -85,B 0,C 180,E1 -16132.69,E2 -16132.69} C_VEL
LIN {X 0,Y 316.268,Z 552.693,A -85,B 0,C 180,E1 -16134.134,E2 -16134.134} C_VEL
LIN {X 0,Y 317.969,Z 539.848,A -85,B 0,C 180,E1 -16135.339,E2 -16135.339} C_VEL
LIN {X 0,Y 317.877,Z 535.146,A -85,B 0,C 180,E1 -16135.771,E2 -16135.771} C_VEL
LIN {X 0,Y 316.105,Z 522.833,A -85,B 0,C 180,E1 -16136.861,E2 -16136.861} C_VEL
LIN {X 0,Y 313.309,Z 509.375,A -85,B 0,C 180,E1 -16137.879,E2 -16137.879} C_VEL
LIN {X 0,Y 309.094,Z 494.31,A -85,B 0,C 180,E1 -16138.839,E2 -16138.839} C_VEL
LIN {X 0,Y 308.179,Z 491.251,A -85,B 0,C 180,E1 -16139.04,E2 -16139.04} C_VEL
LIN {X 0,Y 308.876,Z 481.557,A -85,B 0,C 180,E1 -16142.661,E2 -16142.661} C_VEL
LIN {X 0,Y 309.746,Z 470.902,A -85,B 0,C 180,E1 -16146.807,E2 -16146.807} C_VEL
LIN {X 0,Y 310.509,Z 462.358,A -85,B 0,C 180,E1 -16150.238,E2 -16150.238} C_VEL
LIN {X 0,Y 310.06,Z 457.446,A -85,B 0,C 180,E1 -16152.38,E2 -16152.38} C_VEL
LIN {X 0,Y 308.906,Z 451.312,A -85,B 0,C 180,E1 -16155.147,E2 -16155.147} C_VEL
LIN {X 0,Y 307.415,Z 444.156,A -85,B 0,C 180,E1 -16158.472,E2 -16158.472} C_VEL
LIN {X 0,Y 305.513,Z 436.052,A -85,B 0,C 180,E1 -16162.439,E2 -16162.439} C_VEL
LIN {X 0,Y 305.466,Z 436.051,A -85,B 0,C 180,E1 -16166.483,E2 -16166.483} C_VEL
LIN {X 0,Y 305.461,Z 436.048,A -85,B 0,C 180,E1 -16170.107,E2 -16170.107} C_VEL
LIN {X 0,Y 305.424,Z 436.643,A -85,B 0,C 180,E1 -16170.626,E2 -16170.626} C_VEL
LIN {X 0,Y 305.29,Z 438.715,A -85,B 0,C 180,E1 -16171.231,E2 -16171.231} C_VEL
LIN {X 0,Y 305.073,Z 442.543,A -85,B 0,C 180,E1 -16171.848,E2 -16171.848} C_VEL
LIN {X 0,Y 304.925,Z 448.013,A -85,B 0,C 180,E1 -16172.416,E2 -16172.416} C_VEL
LIN {X 0,Y 304.998,Z 454.007,A -85,B 0,C 180,E1 -16172.953,E2 -16172.953} C_VEL
LIN {X 0,Y 305.723,Z 459.301,A -85,B 0,C 180,E1 -16173.508,E2 -16173.508} C_VEL
LIN {X 0,Y 306.152,Z 460.974,A -85,B 0,C 180,E1 -16173.71,E2 -16173.71} C_VEL
LIN {X 0,Y 308.44,Z 468.822,A -85,B 0,C 180,E1 -16174.708,E2 -16174.708} C_VEL
LIN {X 0,Y 307.971,Z 474.793,A -85,B 0,C 180,E1 -16175.388,E2 -16175.388} C_VEL
LIN {X 0,Y 306.302,Z 487.719,A -85,B 0,C 180,E1 -16177.042,E2 -16177.042} C_VEL
LIN {X 0,Y 304.399,Z 500.646,A -85,B 0,C 180,E1 -16179.031,E2 -16179.031} C_VEL
LIN {X 0,Y 302.843,Z 511.514,A -85,B 0,C 180,E1 -16181.041,E2 -16181.041} C_VEL
LIN {X 0,Y 301.17,Z 522.432,A -85,B 0,C 180,E1 -16183.458,E2 -16183.458} C_VEL
LIN {X 0,Y 300.261,Z 529.842,A -85,B 0,C 180,E1 -16185.427,E2 -16185.427} C_VEL
LIN {X 0,Y 299.236,Z 537.409,A -85,B 0,C 180,E1 -16187.797,E2 -16187.797} C_VEL
LIN {X 0,Y 298.43,Z 544.432,A -85,B 0,C 180,E1 -16190.511,E2 -16190.511} C_VEL
LIN {X 0,Y 297.924,Z 549.939,A -85,B 0,C 180,E1 -16193.226,E2 -16193.226} C_VEL
LIN {X 0,Y 297.797,Z 554.051,A -85,B 0,C 180,E1 -16195.94,E2 -16195.94} C_VEL
LIN {X 0,Y 297.499,Z 556.904,A -85,B 0,C 180,E1 -16198.646,E2 -16198.646} C_VEL
LIN {X 0,Y 297.527,Z 558.544,A -85,B 0,C 180,E1 -16201.353,E2 -16201.353} C_VEL
LIN {X 0,Y 298.046,Z 558.963,A -85,B 0,C 180,E1 -16204.056,E2 -16204.056} C_VEL
LIN {X 0,Y 298.928,Z 558.189,A -85,B 0,C 180,E1 -16206.751,E2 -16206.751} C_VEL
LIN {X 0,Y 299.951,Z 556.251,A -85,B 0,C 180,E1 -16209.44,E2 -16209.44} C_VEL
LIN {X 0,Y 301.338,Z 553.079,A -85,B 0,C 180,E1 -16212.117,E2 -16212.117} C_VEL
LIN {X 0,Y 303.002,Z 548.669,A -85,B 0,C 180,E1 -16214.782,E2 -16214.782} C_VEL
LIN {X 0,Y 305.303,Z 542.818,A -85,B 0,C 180,E1 -16217.413,E2 -16217.413} C_VEL
LIN {X 0,Y 307.365,Z 537.415,A -85,B 0,C 180,E1 -16219.363,E2 -16219.363} C_VEL
LIN {X 0,Y 310.444,Z 529.061,A -85,B 0,C 180,E1 -16221.847,E2 -16221.847} C_VEL
LIN {X 0,Y 313.644,Z 519.64,A -85,B 0,C 180,E1 -16224.138,E2 -16224.138} C_VEL
LIN {X 0,Y 317.247,Z 508.661,A -85,B 0,C 180,E1 -16226.299,E2 -16226.299} C_VEL
LIN {X 0,Y 320.935,Z 496.718,A -85,B 0,C 180,E1 -16228.21,E2 -16228.21} C_VEL
LIN {X 0,Y 323.953,Z 485.197,A -85,B 0,C 180,E1 -16229.798,E2 -16229.798} C_VEL
LIN {X 0,Y 322.185,Z 477.233,A -85,B 0,C 180,E1 -16231.709,E2 -16231.709} C_VEL
LIN {X 0,Y 319.395,Z 469.271,A -85,B 0,C 180,E1 -16234.046,E2 -16234.046} C_VEL
LIN {X 0,Y 316.997,Z 464.225,A -85,B 0,C 180,E1 -16235.946,E2 -16235.946} C_VEL
LIN {X 0,Y 315.444,Z 462.688,A -85,B 0,C 180,E1 -16236.981,E2 -16236.981} C_VEL
LIN {X 0,Y 312.898,Z 460.576,A -85,B 0,C 180,E1 -16238.97,E2 -16238.97} C_VEL
LIN {X 0,Y 310.322,Z 460.007,A -85,B 0,C 180,E1 -16241.637,E2 -16241.637} C_VEL
LIN {X 0,Y 309.334,Z 460.375,A -85,B 0,C 180,E1 -16243.362,E2 -16243.362} C_VEL
LIN {X 0,Y 308.552,Z 462.477,A -85,B 0,C 180,E1 -16245.082,E2 -16245.082} C_VEL
LIN {X 0,Y 308.302,Z 465.375,A -85,B 0,C 180,E1 -16246.853,E2 -16246.853} C_VEL
LIN {X 0,Y 308.513,Z 472.756,A -85,B 0,C 180,E1 -16249.632,E2 -16249.632} C_VEL
LIN {X 0,Y 309.453,Z 476.453,A -85,B 0,C 180,E1 -16251.064,E2 -16251.064} C_VEL
LIN {X 0,Y 310.86,Z 484.727,A -85,B 0,C 180,E1 -16253.273,E2 -16253.273} C_VEL
LIN {X 0,Y 311.991,Z 491.241,A -85,B 0,C 180,E1 -16254.75,E2 -16254.75} C_VEL
LIN {X 0,Y 313.452,Z 502.875,A -85,B 0,C 180,E1 -16256.969,E2 -16256.969} C_VEL
LIN {X 0,Y 314.192,Z 513.815,A -85,B 0,C 180,E1 -16258.782,E2 -16258.782} C_VEL
LIN {X 0,Y 313.995,Z 525.285,A -85,B 0,C 180,E1 -16260.501,E2 -16260.501} C_VEL
LIN {X 0,Y 312.613,Z 537.186,A -85,B 0,C 180,E1 -16262.193,E2 -16262.193} C_VEL
LIN {X 0,Y 311.097,Z 549.994,A -85,B 0,C 180,E1 -16264.222,E2 -16264.222} C_VEL
LIN {X 0,Y 310.529,Z 553.131,A -85,B 0,C 180,E1 -16264.741,E2 -16264.741} C_VEL
LIN {X 0,Y 308.803,Z 559.031,A -85,B 0,C 180,E1 -16265.658,E2 -16265.658} C_VEL
LIN {X 0,Y 306.944,Z 570.73,A -85,B 0,C 180,E1 -16267.093,E2 -16267.093} C_VEL
LIN {X 0,Y 304.869,Z 581.542,A -85,B 0,C 180,E1 -16268.711,E2 -16268.711} C_VEL
LIN {X 0,Y 302.848,Z 592.208,A -85,B 0,C 180,E1 -16270.689,E2 -16270.689} C_VEL
LIN {X 0,Y 301.049,Z 601.129,A -85,B 0,C 180,E1 -16272.719,E2 -16272.719} C_VEL
LIN {X 0,Y 299.716,Z 608.285,A -85,B 0,C 180,E1 -16274.704,E2 -16274.704} C_VEL
LIN {X 0,Y 298.399,Z 615.243,A -85,B 0,C 180,E1 -16277.071,E2 -16277.071} C_VEL
LIN {X 0,Y 297.385,Z 621.469,A -85,B 0,C 180,E1 -16279.791,E2 -16279.791} C_VEL
LIN {X 0,Y 296.95,Z 625,A -85,B 0,C 180,E1 -16281.836,E2 -16281.836} C_VEL
LIN {X 0,Y 296.62,Z 628.441,A -85,B 0,C 180,E1 -16284.562,E2 -16284.562} C_VEL
LIN {X 0,Y 296.572,Z 630.478,A -85,B 0,C 180,E1 -16287.283,E2 -16287.283} C_VEL
LIN {X 0,Y 296.507,Z 631.153,A -85,B 0,C 180,E1 -16290,E2 -16290} C_VEL
LIN {X 0,Y 296.57,Z 630.471,A -85,B 0,C 180,E1 -16292.717,E2 -16292.717} C_VEL
LIN {X 0,Y 296.6,Z 628.43,A -85,B 0,C 180,E1 -16295.439,E2 -16295.439} C_VEL
LIN {X 0,Y 296.915,Z 624.98,A -85,B 0,C 180,E1 -16298.165,E2 -16298.165} C_VEL
LIN {X 0,Y 297.586,Z 620.018,A -85,B 0,C 180,E1 -16300.891,E2 -16300.891} C_VEL
LIN {X 0,Y 298.389,Z 615.203,A -85,B 0,C 180,E1 -16302.93,E2 -16302.93} C_VEL
LIN {X 0,Y 299.655,Z 608.237,A -85,B 0,C 180,E1 -16305.299,E2 -16305.299} C_VEL
LIN {X 0,Y 301.302,Z 599.583,A -85,B 0,C 180,E1 -16307.652,E2 -16307.652} C_VEL
LIN {X 0,Y 303.068,Z 590.511,A -85,B 0,C 180,E1 -16309.648,E2 -16309.648} C_VEL
LIN {X 0,Y 305.21,Z 579.486,A -85,B 0,C 180,E1 -16311.619,E2 -16311.619} C_VEL
LIN {X 0,Y 307.313,Z 568.197,A -85,B 0,C 180,E1 -16313.234,E2 -16313.234} C_VEL
LIN {X 0,Y 309.082,Z 556.892,A -85,B 0,C 180,E1 -16314.559,E2 -16314.559} C_VEL
LIN {X 0,Y 309.985,Z 550.704,A -85,B 0,C 180,E1 -16315.171,E2 -16315.171} C_VEL
LIN {X 0,Y 309.105,Z 538.026,A -85,B 0,C 180,E1 -16316.441,E2 -16316.441} C_VEL
LIN {X 0,Y 307.255,Z 523.962,A -85,B 0,C 180,E1 -16317.629,E2 -16317.629} C_VEL
LIN {X 0,Y 304.885,Z 509.356,A -85,B 0,C 180,E1 -16318.605,E2 -16318.605} C_VEL
LIN {X 0,Y 302.829,Z 500.206,A -85,B 0,C 180,E1 -16319.125,E2 -16319.125} C_VEL
LIN {X 0,Y 299.678,Z 489.768,A -85,B 0,C 180,E1 -16319.763,E2 -16319.763} C_VEL
LIN {X 0,Y 298.593,Z 481.123,A -85,B 0,C 180,E1 -16321.244,E2 -16321.244} C_VEL
LIN {X 0,Y 299.216,Z 474.4,A -85,B 0,C 180,E1 -16325.262,E2 -16325.262} C_VEL
LIN {X 0,Y 299.823,Z 467.741,A -85,B 0,C 180,E1 -16329.327,E2 -16329.327} C_VEL
LIN {X 0,Y 300.582,Z 460.945,A -85,B 0,C 180,E1 -16333.546,E2 -16333.546} C_VEL
LIN {X 0,Y 301.048,Z 456.564,A -85,B 0,C 180,E1 -16336.361,E2 -16336.361} C_VEL
LIN {X 0,Y 301.17,Z 453.578,A -85,B 0,C 180,E1 -16338.309,E2 -16338.309} C_VEL
LIN {X 0,Y 300.724,Z 449.824,A -85,B 0,C 180,E1 -16340.876,E2 -16340.876} C_VEL
LIN {X 0,Y 299.613,Z 443.809,A -85,B 0,C 180,E1 -16345.184,E2 -16345.184} C_VEL
LIN {X 0,Y 299.079,Z 440.342,A -85,B 0,C 180,E1 -16347.775,E2 -16347.775} C_VEL
LIN {X 0,Y 298.525,Z 436.929,A -85,B 0,C 180,E1 -16350.482,E2 -16350.482} C_VEL
LIN {X 0,Y 298.487,Z 436.916,A -85,B 0,C 180,E1 -16354.924,E2 -16354.924} C_VEL
LIN {X 0,Y 298.451,Z 436.914,A -85,B 0,C 180,E1 -16359.315,E2 -16359.315} C_VEL
LIN {X 0,Y 298.54,Z 436.924,A -85,B 0,C 180,E1 -16362.18,E2 -16362.18} C_VEL
LIN {X 0,Y 298.595,Z 436.895,A -85,B 0,C 180,E1 -16364.995,E2 -16364.995} C_VEL
LIN {X 0,Y 298.585,Z 436.912,A -85,B 0,C 180,E1 -16369.146,E2 -16369.146} C_VEL
LIN {X 0,Y 298.778,Z 436.892,A -85,B 0,C 180,E1 -16373.246,E2 -16373.246} C_VEL
LIN {X 0,Y 298.925,Z 436.866,A -85,B 0,C 180,E1 -16378.653,E2 -16378.653} C_VEL
LIN {X 0,Y 298.925,Z 436.867,A -85,B 0,C 180,E1 -16381.347,E2 -16381.347} C_VEL
LIN {X 0,Y 298.8,Z 436.888,A -85,B 0,C 180,E1 -16386.754,E2 -16386.754} C_VEL
LIN {X 0,Y 298.682,Z 436.891,A -85,B 0,C 180,E1 -16389.481,E2 -16389.481} C_VEL
LIN {X 0,Y 298.554,Z 436.906,A -85,B 0,C 180,E1 -16393.615,E2 -16393.615} C_VEL
LIN {X 0,Y 298.55,Z 436.925,A -85,B 0,C 180,E1 -16396.409,E2 -16396.409} C_VEL
LIN {X 0,Y 298.499,Z 436.92,A -85,B 0,C 180,E1 -16399.647,E2 -16399.647} C_VEL
LIN {X 0,Y 298.43,Z 436.928,A -85,B 0,C 180,E1 -16403.6,E2 -16403.6} C_VEL
LIN {X 0,Y 298.491,Z 436.919,A -85,B 0,C 180,E1 -16406.574,E2 -16406.574} C_VEL
LIN {X 0,Y 298.422,Z 436.931,A -85,B 0,C 180,E1 -16409.641,E2 -16409.641} C_VEL
LIN {X 0,Y 298.397,Z 436.935,A -85,B 0,C 180,E1 -16412.8,E2 -16412.8} C_VEL
LIN {X 0,Y 298.449,Z 437.006,A -85,B 0,C 180,E1 -16416.88,E2 -16416.88} C_VEL
LIN {X 0,Y 299.994,Z 443.466,A -85,B 0,C 180,E1 -16420.109,E2 -16420.109} C_VEL
LIN {X 0,Y 301.455,Z 449.808,A -85,B 0,C 180,E1 -16423.176,E2 -16423.176} C_VEL
LIN {X 0,Y 302.98,Z 457.817,A -85,B 0,C 180,E1 -16426.902,E2 -16426.902} C_VEL
LIN {X 0,Y 303.703,Z 463.869,A -85,B 0,C 180,E1 -16429.613,E2 -16429.613} C_VEL
LIN {X 0,Y 302.859,Z 473.005,A -85,B 0,C 180,E1 -16433.306,E2 -16433.306} C_VEL
LIN {X 0,Y 302.093,Z 482.051,A -85,B 0,C 180,E1 -16436.879,E2 -16436.879} C_VEL
LIN {X 0,Y 301.405,Z 491.327,A -85,B 0,C 180,E1 -16440.391,E2 -16440.391} C_VEL
LIN {X 0,Y 306.019,Z 507.139,A -85,B 0,C 180,E1 -16441.414,E2 -16441.414} C_VEL
LIN {X 0,Y 309.085,Z 520.951,A -85,B 0,C 180,E1 -16442.472,E2 -16442.472} C_VEL
LIN {X 0,Y 311.035,Z 534.064,A -85,B 0,C 180,E1 -16443.64,E2 -16443.64} C_VEL
LIN {X 0,Y 311.491,Z 539.25,A -85,B 0,C 180,E1 -16444.15,E2 -16444.15} C_VEL
LIN {X 0,Y 309.912,Z 551.756,A -85,B 0,C 180,E1 -16445.337,E2 -16445.337} C_VEL
LIN {X 0,Y 308.061,Z 562.971,A -85,B 0,C 180,E1 -16446.647,E2 -16446.647} C_VEL
LIN {X 0,Y 305.902,Z 574.226,A -85,B 0,C 180,E1 -16448.256,E2 -16448.256} C_VEL
LIN {X 0,Y 303.953,Z 584.444,A -85,B 0,C 180,E1 -16450.059,E2 -16450.059} C_VEL
LIN {X 0,Y 301.966,Z 593.675,A -85,B 0,C 180,E1 -16452.038,E2 -16452.038} C_VEL
LIN {X 0,Y 300.483,Z 601.331,A -85,B 0,C 180,E1 -16454.049,E2 -16454.049} C_VEL
LIN {X 0,Y 299.485,Z 606.689,A -85,B 0,C 180,E1 -16455.735,E2 -16455.735} C_VEL
LIN {X 0,Y 298.325,Z 612.142,A -85,B 0,C 180,E1 -16457.759,E2 -16457.759} C_VEL
LIN {X 0,Y 297.373,Z 617.85,A -85,B 0,C 180,E1 -16460.477,E2 -16460.477} C_VEL
LIN {X 0,Y 296.85,Z 622.001,A -85,B 0,C 180,E1 -16463.202,E2 -16463.202} C_VEL
LIN {X 0,Y 296.555,Z 624.718,A -85,B 0,C 180,E1 -16465.923,E2 -16465.923} C_VEL
LIN {X 0,Y 296.458,Z 626.079,A -85,B 0,C 180,E1 -16468.642,E2 -16468.642} C_VEL
LIN {X 0,Y 296.457,Z 626.111,A -85,B 0,C 180,E1 -16471.358,E2 -16471.358} C_VEL
LIN {X 0,Y 296.532,Z 625.625,A -85,B 0,C 180,E1 -16472.717,E2 -16472.717} C_VEL
LIN {X 0,Y 296.621,Z 623.643,A -85,B 0,C 180,E1 -16475.438,E2 -16475.438} C_VEL
LIN {X 0,Y 297.054,Z 620.277,A -85,B 0,C 180,E1 -16478.161,E2 -16478.161} C_VEL
LIN {X 0,Y 297.767,Z 615.425,A -85,B 0,C 180,E1 -16480.884,E2 -16480.884} C_VEL
LIN {X 0,Y 298.611,Z 610.721,A -85,B 0,C 180,E1 -16482.92,E2 -16482.92} C_VEL
LIN {X 0,Y 300.109,Z 603.901,A -85,B 0,C 180,E1 -16485.275,E2 -16485.275} C_VEL
LIN {X 0,Y 301.7,Z 595.438,A -85,B 0,C 180,E1 -16487.628,E2 -16487.628} C_VEL
LIN {X 0,Y 303.53,Z 586.586,A -85,B 0,C 180,E1 -16489.617,E2 -16489.617} C_VEL
LIN {X 0,Y 305.611,Z 575.869,A -85,B 0,C 180,E1 -16491.589,E2 -16491.589} C_VEL
LIN {X 0,Y 307.751,Z 564.994,A -85,B 0,C 180,E1 -16493.199,E2 -16493.199} C_VEL
LIN {X 0,Y 309.859,Z 552.249,A -85,B 0,C 180,E1 -16494.722,E2 -16494.722} C_VEL
LIN {X 0,Y 311.519,Z 540.128,A -85,B 0,C 180,E1 -16495.878,E2 -16495.878} C_VEL
LIN {X 0,Y 310.684,Z 530.659,A -85,B 0,C 180,E1 -16496.788,E2 -16496.788} C_VEL
LIN {X 0,Y 308.234,Z 516.344,A -85,B 0,C 180,E1 -16498.013,E2 -16498.013} C_VEL
LIN {X 0,Y 304.641,Z 502.033,A -85,B 0,C 180,E1 -16499.053,E2 -16499.053} C_VEL
LIN {X 0,Y 301.418,Z 491.245,A -85,B 0,C 180,E1 -16499.756,E2 -16499.756} C_VEL
LIN {X 0,Y 302.174,Z 481.6,A -85,B 0,C 180,E1 -16503.421,E2 -16503.421} C_VEL
LIN {X 0,Y 302.94,Z 472.28,A -85,B 0,C 180,E1 -16507.098,E2 -16507.098} C_VEL
LIN {X 0,Y 303.711,Z 464.235,A -85,B 0,C 180,E1 -16510.386,E2 -16510.386} C_VEL
LIN {X 0,Y 303.361,Z 460.046,A -85,B 0,C 180,E1 -16512.21,E2 -16512.21} C_VEL
LIN {X 0,Y 301.981,Z 452.509,A -85,B 0,C 180,E1 -16515.718,E2 -16515.718} C_VEL
LIN {X 0,Y 300.481,Z 445.401,A -85,B 0,C 180,E1 -16519.088,E2 -16519.088} C_VEL
LIN {X 0,Y 298.925,Z 438.836,A -85,B 0,C 180,E1 -16522.317,E2 -16522.317} C_VEL
LIN {X 0,Y 298.464,Z 436.927,A -85,B 0,C 180,E1 -16523.311,E2 -16523.311} C_VEL
LIN {X 0,Y 298.397,Z 436.937,A -85,B 0,C 180,E1 -16527.2,E2 -16527.2} C_VEL
LIN {X 0,Y 298.486,Z 436.962,A -85,B 0,C 180,E1 -16531.104,E2 -16531.104} C_VEL
LIN {X 0,Y 303.502,Z 452.314,A -85,B 0,C 180,E1 -16532.7,E2 -16532.7} C_VEL
LIN {X 0,Y 306.152,Z 460.974,A -85,B 0,C 180,E1 -16533.71,E2 -16533.71} C_VEL
LIN {X 0,Y 306.621,Z 464.325,A -85,B 0,C 180,E1 -16534.095,E2 -16534.095} C_VEL
LIN {X 0,Y 306.33,Z 467.774,A -85,B 0,C 180,E1 -16534.455,E2 -16534.455} C_VEL
LIN {X 0,Y 304.311,Z 474.515,A -85,B 0,C 180,E1 -16535.132,E2 -16535.132} C_VEL
LIN {X 0,Y 300.304,Z 484.593,A -85,B 0,C 180,E1 -16536.234,E2 -16536.234} C_VEL
LIN {X 0,Y 299.484,Z 487.867,A -85,B 0,C 180,E1 -16536.673,E2 -16536.673} C_VEL
LIN {X 0,Y 297.662,Z 499.897,A -85,B 0,C 180,E1 -16538.533,E2 -16538.533} C_VEL
LIN {X 0,Y 296.046,Z 511.014,A -85,B 0,C 180,E1 -16540.588,E2 -16540.588} C_VEL
LIN {X 0,Y 294.318,Z 521.71,A -85,B 0,C 180,E1 -16542.951,E2 -16542.951} C_VEL
LIN {X 0,Y 293.362,Z 529.754,A -85,B 0,C 180,E1 -16545.076,E2 -16545.076} C_VEL
LIN {X 0,Y 292.247,Z 537.499,A -85,B 0,C 180,E1 -16547.5,E2 -16547.5} C_VEL
LIN {X 0,Y 291.414,Z 544.673,A -85,B 0,C 180,E1 -16550.281,E2 -16550.281} C_VEL
LIN {X 0,Y 290.889,Z 550.31,A -85,B 0,C 180,E1 -16553.061,E2 -16553.061} C_VEL
LIN {X 0,Y 290.741,Z 554.562,A -85,B 0,C 180,E1 -16555.841,E2 -16555.841} C_VEL
LIN {X 0,Y 290.459,Z 557.562,A -85,B 0,C 180,E1 -16558.613,E2 -16558.613} C_VEL
LIN {X 0,Y 290.487,Z 559.343,A -85,B 0,C 180,E1 -16561.386,E2 -16561.386} C_VEL
LIN {X 0,Y 291.029,Z 559.905,A -85,B 0,C 180,E1 -16564.154,E2 -16564.154} C_VEL
LIN {X 0,Y 291.956,Z 559.251,A -85,B 0,C 180,E1 -16566.913,E2 -16566.913} C_VEL
LIN {X 0,Y 293.047,Z 557.435,A -85,B 0,C 180,E1 -16569.664,E2 -16569.664} C_VEL
LIN {X 0,Y 294.514,Z 554.436,A -85,B 0,C 180,E1 -16572.402,E2 -16572.402} C_VEL
LIN {X 0,Y 296.301,Z 550.185,A -85,B 0,C 180,E1 -16575.124,E2 -16575.124} C_VEL
LIN {X 0,Y 298.758,Z 544.564,A -85,B 0,C 180,E1 -16577.807,E2 -16577.807} C_VEL
LIN {X 0,Y 300.935,Z 539.34,A -85,B 0,C 180,E1 -16579.793,E2 -16579.793} C_VEL
LIN {X 0,Y 304.195,Z 531.269,A -85,B 0,C 180,E1 -16582.319,E2 -16582.319} C_VEL
LIN {X 0,Y 308.09,Z 520.829,A -85,B 0,C 180,E1 -16584.962,E2 -16584.962} C_VEL
LIN {X 0,Y 311.951,Z 509.956,A -85,B 0,C 180,E1 -16587.143,E2 -16587.143} C_VEL
LIN {X 0,Y 315.642,Z 498.924,A -85,B 0,C 180,E1 -16588.965,E2 -16588.965} C_VEL
LIN {X 0,Y 318.697,Z 488.465,A -85,B 0,C 180,E1 -16590.478,E2 -16590.478} C_VEL
LIN {X 0,Y 317.551,Z 482.178,A -85,B 0,C 180,E1 -16592.084,E2 -16592.084} C_VEL
LIN {X 0,Y 315.24,Z 474.635,A -85,B 0,C 180,E1 -16594.423,E2 -16594.423} C_VEL
LIN {X 0,Y 313.412,Z 470.236,A -85,B 0,C 180,E1 -16596.17,E2 -16596.17} C_VEL
LIN {X 0,Y 311.302,Z 468.213,A -85,B 0,C 180,E1 -16597.799,E2 -16597.799} C_VEL
LIN {X 0,Y 309.404,Z 466.941,A -85,B 0,C 180,E1 -16599.495,E2 -16599.495} C_VEL
LIN {X 0,Y 307.699,Z 466.58,A -85,B 0,C 180,E1 -16601.481,E2 -16601.481} C_VEL
LIN {X 0,Y 306.915,Z 466.763,A -85,B 0,C 180,E1 -16602.881,E2 -16602.881} C_VEL
LIN {X 0,Y 305.975,Z 468.605,A -85,B 0,C 180,E1 -16604.598,E2 -16604.598} C_VEL
LIN {X 0,Y 305.511,Z 471.372,A -85,B 0,C 180,E1 -16606.36,E2 -16606.36} C_VEL
LIN {X 0,Y 305.379,Z 479.154,A -85,B 0,C 180,E1 -16609.417,E2 -16609.417} C_VEL
LIN {X 0,Y 305.98,Z 482.798,A -85,B 0,C 180,E1 -16610.771,E2 -16610.771} C_VEL
LIN {X 0,Y 306.862,Z 490.097,A -85,B 0,C 180,E1 -16612.776,E2 -16612.776} C_VEL
LIN {X 0,Y 307.69,Z 497.46,A -85,B 0,C 180,E1 -16614.476,E2 -16614.476} C_VEL
LIN {X 0,Y 308.628,Z 508.19,A -85,B 0,C 180,E1 -16616.628,E2 -16616.628} C_VEL
LIN {X 0,Y 308.784,Z 518.654,A -85,B 0,C 180,E1 -16618.434,E2 -16618.434} C_VEL
LIN {X 0,Y 307.999,Z 530.442,A -85,B 0,C 180,E1 -16620.295,E2 -16620.295} C_VEL
LIN {X 0,Y 305.42,Z 546.414,A -85,B 0,C 180,E1 -16622.784,E2 -16622.784} C_VEL
LIN {X 0,Y 304.253,Z 554.319,A -85,B 0,C 180,E1 -16624.17,E2 -16624.17} C_VEL
LIN {X 0,Y 301.944,Z 561.67,A -85,B 0,C 180,E1 -16625.414,E2 -16625.414} C_VEL
LIN {X 0,Y 299.956,Z 573.024,A -85,B 0,C 180,E1 -16626.893,E2 -16626.893} C_VEL
LIN {X 0,Y 297.857,Z 583.438,A -85,B 0,C 180,E1 -16628.548,E2 -16628.548} C_VEL
LIN {X 0,Y 295.773,Z 593.777,A -85,B 0,C 180,E1 -16630.57,E2 -16630.57} C_VEL
LIN {X 0,Y 293.982,Z 602.287,A -85,B 0,C 180,E1 -16632.613,E2 -16632.613} C_VEL
LIN {X 0,Y 292.423,Z 610.393,A -85,B 0,C 180,E1 -16635.027,E2 -16635.027} C_VEL
LIN {X 0,Y 291.074,Z 616.906,A -85,B 0,C 180,E1 -16637.449,E2 -16637.449} C_VEL
LIN {X 0,Y 290.167,Z 622.665,A -85,B 0,C 180,E1 -16640.239,E2 -16640.239} C_VEL
LIN {X 0,Y 289.67,Z 626.843,A -85,B 0,C 180,E1 -16643.032,E2 -16643.032} C_VEL
LIN {X 0,Y 289.471,Z 629.572,A -85,B 0,C 180,E1 -16645.823,E2 -16645.823} C_VEL
LIN {X 0,Y 289.437,Z 630.927,A -85,B 0,C 180,E1 -16648.609,E2 -16648.609} C_VEL
LIN {X 0,Y 289.437,Z 630.923,A -85,B 0,C 180,E1 -16651.391,E2 -16651.391} C_VEL
LIN {X 0,Y 289.473,Z 630.413,A -85,B 0,C 180,E1 -16652.783,E2 -16652.783} C_VEL
LIN {X 0,Y 289.516,Z 628.371,A -85,B 0,C 180,E1 -16655.572,E2 -16655.572} C_VEL
LIN {X 0,Y 289.864,Z 624.921,A -85,B 0,C 180,E1 -16658.365,E2 -16658.365} C_VEL
LIN {X 0,Y 290.572,Z 619.959,A -85,B 0,C 180,E1 -16661.157,E2 -16661.157} C_VEL
LIN {X 0,Y 291.443,Z 615.145,A -85,B 0,C 180,E1 -16663.243,E2 -16663.243} C_VEL
LIN {X 0,Y 292.759,Z 608.269,A -85,B 0,C 180,E1 -16665.64,E2 -16665.64} C_VEL
LIN {X 0,Y 294.49,Z 599.526,A -85,B 0,C 180,E1 -16668.074,E2 -16668.074} C_VEL
LIN {X 0,Y 296.364,Z 590.457,A -85,B 0,C 180,E1 -16670.112,E2 -16670.112} C_VEL
LIN {X 0,Y 298.601,Z 579.434,A -85,B 0,C 180,E1 -16672.122,E2 -16672.122} C_VEL
LIN {X 0,Y 300.794,Z 568.148,A -85,B 0,C 180,E1 -16673.769,E2 -16673.769} C_VEL
LIN {X 0,Y 302.776,Z 555.889,A -85,B 0,C 180,E1 -16675.218,E2 -16675.218} C_VEL
LIN {X 0,Y 303.385,Z 550.799,A -85,B 0,C 180,E1 -16675.744,E2 -16675.744} C_VEL
LIN {X 0,Y 302.486,Z 537.989,A -85,B 0,C 180,E1 -16677.066,E2 -16677.066} C_VEL
LIN {X 0,Y 300.708,Z 523.787,A -85,B 0,C 180,E1 -16678.294,E2 -16678.294} C_VEL
LIN {X 0,Y 298.402,Z 509.338,A -85,B 0,C 180,E1 -16679.287,E2 -16679.287} C_VEL
LIN {X 0,Y 296.154,Z 500.075,A -85,B 0,C 180,E1 -16679.852,E2 -16679.852} C_VEL
LIN {X 0,Y 292.895,Z 489.753,A -85,B 0,C 180,E1 -16680.537,E2 -16680.537} C_VEL
LIN {X 0,Y 291.664,Z 479.511,A -85,B 0,C 180,E1 -16682.398,E2 -16682.398} C_VEL
LIN {X 0,Y 292.138,Z 474.845,A -85,B 0,C 180,E1 -16685.266,E2 -16685.266} C_VEL
LIN {X 0,Y 292.836,Z 467.516,A -85,B 0,C 180,E1 -16689.826,E2 -16689.826} C_VEL
LIN {X 0,Y 293.597,Z 460.856,A -85,B 0,C 180,E1 -16694.1,E2 -16694.1} C_VEL
LIN {X 0,Y 294.066,Z 456.377,A -85,B 0,C 180,E1 -16697.018,E2 -16697.018} C_VEL
LIN {X 0,Y 293.917,Z 452.33,A -85,B 0,C 180,E1 -16699.789,E2 -16699.789} C_VEL
LIN {X 0,Y 293.082,Z 447.614,A -85,B 0,C 180,E1 -16703.167,E2 -16703.167} C_VEL
LIN {X 0,Y 292.202,Z 442.046,A -85,B 0,C 180,E1 -16707.332,E2 -16707.332} C_VEL
LIN {X 0,Y 291.467,Z 437.808,A -85,B 0,C 180,E1 -16710.681,E2 -16710.681} C_VEL
LIN {X 0,Y 291.417,Z 437.791,A -85,B 0,C 180,E1 -16714.272,E2 -16714.272} C_VEL
LIN {X 0,Y 291.383,Z 437.812,A -85,B 0,C 180,E1 -16717.3,E2 -16717.3} C_VEL
LIN {X 0,Y 291.459,Z 437.788,A -85,B 0,C 180,E1 -16720.27,E2 -16720.27} C_VEL
LIN {X 0,Y 291.556,Z 437.773,A -85,B 0,C 180,E1 -16724.624,E2 -16724.624} C_VEL
LIN {X 0,Y 291.531,Z 437.794,A -85,B 0,C 180,E1 -16728.88,E2 -16728.88} C_VEL
LIN {X 0,Y 291.657,Z 437.76,A -85,B 0,C 180,E1 -16731.687,E2 -16731.687} C_VEL
LIN {X 0,Y 291.626,Z 437.784,A -85,B 0,C 180,E1 -16734.468,E2 -16734.468} C_VEL
LIN {X 0,Y 291.891,Z 437.741,A -85,B 0,C 180,E1 -16738.62,E2 -16738.62} C_VEL
LIN {X 0,Y 291.891,Z 437.743,A -85,B 0,C 180,E1 -16741.38,E2 -16741.38} C_VEL
LIN {X 0,Y 291.748,Z 437.763,A -85,B 0,C 180,E1 -16746.918,E2 -16746.918} C_VEL
LIN {X 0,Y 291.631,Z 437.771,A -85,B 0,C 180,E1 -16749.712,E2 -16749.712} C_VEL
LIN {X 0,Y 291.523,Z 437.781,A -85,B 0,C 180,E1 -16753.95,E2 -16753.95} C_VEL
LIN {X 0,Y 291.488,Z 437.802,A -85,B 0,C 180,E1 -16756.818,E2 -16756.818} C_VEL
LIN {X 0,Y 291.452,Z 437.8,A -85,B 0,C 180,E1 -16759.875,E2 -16759.875} C_VEL
LIN {X 0,Y 291.385,Z 437.811,A -85,B 0,C 180,E1 -16764.207,E2 -16764.207} C_VEL
LIN {X 0,Y 291.424,Z 437.801,A -85,B 0,C 180,E1 -16767.272,E2 -16767.272} C_VEL
LIN {X 0,Y 291.339,Z 437.813,A -85,B 0,C 180,E1 -16770.437,E2 -16770.437} C_VEL
LIN {X 0,Y 291.346,Z 437.815,A -85,B 0,C 180,E1 -16773.698,E2 -16773.698} C_VEL
LIN {X 0,Y 291.382,Z 437.88,A -85,B 0,C 180,E1 -16775.903,E2 -16775.903} C_VEL
LIN {X 0,Y 293.02,Z 444.365,A -85,B 0,C 180,E1 -16779.277,E2 -16779.277} C_VEL
LIN {X 0,Y 294.659,Z 451.58,A -85,B 0,C 180,E1 -16782.83,E2 -16782.83} C_VEL
LIN {X 0,Y 296.083,Z 459.238,A -85,B 0,C 180,E1 -16786.499,E2 -16786.499} C_VEL
LIN {X 0,Y 296.754,Z 463.544,A -85,B 0,C 180,E1 -16788.462,E2 -16788.462} C_VEL
LIN {X 0,Y 296.79,Z 467.676,A -85,B 0,C 180,E1 -16790.256,E2 -16790.256} C_VEL
LIN {X 0,Y 295.718,Z 478.19,A -85,B 0,C 180,E1 -16794.535,E2 -16794.535} C_VEL
LIN {X 0,Y 294.945,Z 488.001,A -85,B 0,C 180,E1 -16798.384,E2 -16798.384} C_VEL
LIN {X 0,Y 294.672,Z 491.348,A -85,B 0,C 180,E1 -16799.647,E2 -16799.647} C_VEL
LIN {X 0,Y 299.456,Z 507.666,A -85,B 0,C 180,E1 -16800.751,E2 -16800.751} C_VEL
LIN {X 0,Y 302.497,Z 521.29,A -85,B 0,C 180,E1 -16801.84,E2 -16801.84} C_VEL
LIN {X 0,Y 304.468,Z 534.716,A -85,B 0,C 180,E1 -16803.078,E2 -16803.078} C_VEL
LIN {X 0,Y 304.989,Z 539.562,A -85,B 0,C 180,E1 -16803.582,E2 -16803.582} C_VEL
LIN {X 0,Y 303.372,Z 552.442,A -85,B 0,C 180,E1 -16804.844,E2 -16804.844} C_VEL
LIN {X 0,Y 301.343,Z 564.285,A -85,B 0,C 180,E1 -16806.277,E2 -16806.277} C_VEL
LIN {X 0,Y 299.088,Z 575.315,A -85,B 0,C 180,E1 -16807.916,E2 -16807.916} C_VEL
LIN {X 0,Y 296.895,Z 586.138,A -85,B 0,C 180,E1 -16809.926,E2 -16809.926} C_VEL
LIN {X 0,Y 294.897,Z 595.074,A -85,B 0,C 180,E1 -16811.952,E2 -16811.952} C_VEL
LIN {X 0,Y 293.431,Z 602.512,A -85,B 0,C 180,E1 -16814.012,E2 -16814.012} C_VEL
LIN {X 0,Y 292.16,Z 608.71,A -85,B 0,C 180,E1 -16816.081,E2 -16816.081} C_VEL
LIN {X 0,Y 291.095,Z 613.792,A -85,B 0,C 180,E1 -16818.158,E2 -16818.158} C_VEL
LIN {X 0,Y 290.177,Z 619.119,A -85,B 0,C 180,E1 -16820.942,E2 -16820.942} C_VEL
LIN {X 0,Y 289.769,Z 622.06,A -85,B 0,C 180,E1 -16823.035,E2 -16823.035} C_VEL
LIN {X 0,Y 289.461,Z 624.777,A -85,B 0,C 180,E1 -16825.823,E2 -16825.823} C_VEL
LIN {X 0,Y 289.382,Z 626.138,A -85,B 0,C 180,E1 -16828.608,E2 -16828.608} C_VEL
LIN {X 0,Y 289.381,Z 626.169,A -85,B 0,C 180,E1 -16831.392,E2 -16831.392} C_VEL
LIN {X 0,Y 289.454,Z 624.862,A -85,B 0,C 180,E1 -16834.177,E2 -16834.177} C_VEL
LIN {X 0,Y 289.734,Z 622.195,A -85,B 0,C 180,E1 -16836.966,E2 -16836.966} C_VEL
LIN {X 0,Y 290.333,Z 618.102,A -85,B 0,C 180,E1 -16839.756,E2 -16839.756} C_VEL
LIN {X 0,Y 291.287,Z 612.452,A -85,B 0,C 180,E1 -16842.542,E2 -16842.542} C_VEL
LIN {X 0,Y 292.787,Z 606.063,A -85,B 0,C 180,E1 -16844.954,E2 -16844.954} C_VEL
LIN {X 0,Y 294.386,Z 597.963,A -85,B 0,C 180,E1 -16847.411,E2 -16847.411} C_VEL
LIN {X 0,Y 296.135,Z 589.806,A -85,B 0,C 180,E1 -16849.406,E2 -16849.406} C_VEL
LIN {X 0,Y 298.24,Z 579.749,A -85,B 0,C 180,E1 -16851.423,E2 -16851.423} C_VEL
LIN {X 0,Y 300.512,Z 568.491,A -85,B 0,C 180,E1 -16853.244,E2 -16853.244} C_VEL
LIN {X 0,Y 302.785,Z 556.277,A -85,B 0,C 180,E1 -16854.83,E2 -16854.83} C_VEL
LIN {X 0,Y 304.706,Z 543.59,A -85,B 0,C 180,E1 -16856.152,E2 -16856.152} C_VEL
LIN {X 0,Y 304.965,Z 538.776,A -85,B 0,C 180,E1 -16856.609,E2 -16856.609} C_VEL
LIN {X 0,Y 303.321,Z 526.203,A -85,B 0,C 180,E1 -16857.842,E2 -16857.842} C_VEL
LIN {X 0,Y 300.789,Z 513.09,A -85,B 0,C 180,E1 -16858.949,E2 -16858.949} C_VEL
LIN {X 0,Y 297.129,Z 499.387,A -85,B 0,C 180,E1 -16859.952,E2 -16859.952} C_VEL
LIN {X 0,Y 294.699,Z 491.239,A -85,B 0,C 180,E1 -16860.505,E2 -16860.505} C_VEL
LIN {X 0,Y 295.555,Z 480.189,A -85,B 0,C 180,E1 -16864.799,E2 -16864.799} C_VEL
LIN {X 0,Y 296.42,Z 471.022,A -85,B 0,C 180,E1 -16868.517,E2 -16868.517} C_VEL
LIN {X 0,Y 296.907,Z 465.616,A -85,B 0,C 180,E1 -16870.759,E2 -16870.759} C_VEL
LIN {X 0,Y 296.447,Z 461.3,A -85,B 0,C 180,E1 -16872.698,E2 -16872.698} C_VEL
LIN {X 0,Y 295.071,Z 453.673,A -85,B 0,C 180,E1 -16876.312,E2 -16876.312} C_VEL
LIN {X 0,Y 293.407,Z 446.113,A -85,B 0,C 180,E1 -16880.041,E2 -16880.041} C_VEL
LIN {X 0,Y 292.047,Z 440.283,A -85,B 0,C 180,E1 -16883.014,E2 -16883.014} C_VEL
LIN {X 0,Y 291.38,Z 437.816,A -85,B 0,C 180,E1 -16884.31,E2 -16884.31} C_VEL
LIN {X 0,Y 291.374,Z 437.817,A -85,B 0,C 180,E1 -16887.951,E2 -16887.951} C_VEL
LIN {X 0,Y 291.444,Z 437.944,A -85,B 0,C 180,E1 -16890.667,E2 -16890.667} C_VEL
LIN {X 0,Y 296.472,Z 453.208,A -85,B 0,C 180,E1 -16892.311,E2 -16892.311} C_VEL
LIN {X 0,Y 300.809,Z 467.62,A -85,B 0,C 180,E1 -16894.091,E2 -16894.091} C_VEL
LIN {X 0,Y 301.562,Z 470.326,A -85,B 0,C 180,E1 -16894.459,E2 -16894.459} C_VEL
LIN {X 0,Y 300.583,Z 479.811,A -85,B 0,C 180,E1 -16895.589,E2 -16895.589} C_VEL
LIN {X 0,Y 299.484,Z 487.867,A -85,B 0,C 180,E1 -16896.673,E2 -16896.673} C_VEL
LIN {X 0,Y 298.106,Z 492.554,A -85,B 0,C 180,E1 -16897.314,E2 -16897.314} C_VEL
LIN {X 0,Y 291.094,Z 505.698,A -85,B 0,C 180,E1 -16899.23,E2 -16899.23} C_VEL
LIN {X 0,Y 289.444,Z 509.874,A -85,B 0,C 180,E1 -16899.989,E2 -16899.989} C_VEL
LIN {X 0,Y 289.139,Z 511.234,A -85,B 0,C 180,E1 -16900.265,E2 -16900.265} C_VEL
LIN {X 0,Y 287.494,Z 521.037,A -85,B 0,C 180,E1 -16902.437,E2 -16902.437} C_VEL
LIN {X 0,Y 286.457,Z 529.614,A -85,B 0,C 180,E1 -16904.708,E2 -16904.708} C_VEL
LIN {X 0,Y 285.279,Z 537.5,A -85,B 0,C 180,E1 -16907.19,E2 -16907.19} C_VEL
LIN {X 0,Y 284.398,Z 544.86,A -85,B 0,C 180,E1 -16910.039,E2 -16910.039} C_VEL
LIN {X 0,Y 283.858,Z 550.663,A -85,B 0,C 180,E1 -16912.889,E2 -16912.889} C_VEL
LIN {X 0,Y 283.686,Z 555.073,A -85,B 0,C 180,E1 -16915.738,E2 -16915.738} C_VEL
LIN {X 0,Y 283.42,Z 558.211,A -85,B 0,C 180,E1 -16918.579,E2 -16918.579} C_VEL
LIN {X 0,Y 283.448,Z 560.117,A -85,B 0,C 180,E1 -16921.421,E2 -16921.421} C_VEL
LIN {X 0,Y 284.013,Z 560.798,A -85,B 0,C 180,E1 -16924.257,E2 -16924.257} C_VEL
LIN {X 0,Y 284.987,Z 560.285,A -85,B 0,C 180,E1 -16927.083,E2 -16927.083} C_VEL
LIN {X 0,Y 286.17,Z 558.636,A -85,B 0,C 180,E1 -16929.899,E2 -16929.899} C_VEL
LIN {X 0,Y 287.71,Z 555.8,A -85,B 0,C 180,E1 -16932.7,E2 -16932.7} C_VEL
LIN {X 0,Y 289.63,Z 551.761,A -85,B 0,C 180,E1 -16935.481,E2 -16935.481} C_VEL
LIN {X 0,Y 292.238,Z 546.336,A -85,B 0,C 180,E1 -16938.218,E2 -16938.218} C_VEL
LIN {X 0,Y 294.533,Z 541.364,A -85,B 0,C 180,E1 -16940.242,E2 -16940.242} C_VEL
LIN {X 0,Y 297.8,Z 533.946,A -85,B 0,C 180,E1 -16942.702,E2 -16942.702} C_VEL
LIN {X 0,Y 301.549,Z 524.767,A -85,B 0,C 180,E1 -16945.172,E2 -16945.172} C_VEL
LIN {X 0,Y 305.524,Z 514.684,A -85,B 0,C 180,E1 -16947.391,E2 -16947.391} C_VEL
LIN {X 0,Y 310.031,Z 502.625,A -85,B 0,C 180,E1 -16949.541,E2 -16949.541} C_VEL
LIN {X 0,Y 313.54,Z 491.719,A -85,B 0,C 180,E1 -16951.195,E2 -16951.195} C_VEL
LIN {X 0,Y 312.736,Z 486.51,A -85,B 0,C 180,E1 -16952.639,E2 -16952.639} C_VEL
LIN {X 0,Y 311.079,Z 479.95,A -85,B 0,C 180,E1 -16954.814,E2 -16954.814} C_VEL
LIN {X 0,Y 309.952,Z 476.789,A -85,B 0,C 180,E1 -16956.124,E2 -16956.124} C_VEL
LIN {X 0,Y 307.81,Z 474.332,A -85,B 0,C 180,E1 -16958.059,E2 -16958.059} C_VEL
LIN {X 0,Y 305.785,Z 473.23,A -85,B 0,C 180,E1 -16960.056,E2 -16960.056} C_VEL
LIN {X 0,Y 304.256,Z 473.166,A -85,B 0,C 180,E1 -16962.339,E2 -16962.339} C_VEL
LIN {X 0,Y 303.247,Z 474.624,A -85,B 0,C 180,E1 -16964.073,E2 -16964.073} C_VEL
LIN {X 0,Y 302.467,Z 477.795,A -85,B 0,C 180,E1 -16966.08,E2 -16966.08} C_VEL
LIN {X 0,Y 301.964,Z 484.635,A -85,B 0,C 180,E1 -16968.859,E2 -16968.859} C_VEL
LIN {X 0,Y 302.295,Z 487.786,A -85,B 0,C 180,E1 -16970.104,E2 -16970.104} C_VEL
LIN {X 0,Y 302.762,Z 494.71,A -85,B 0,C 180,E1 -16972.115,E2 -16972.115} C_VEL
LIN {X 0,Y 303.169,Z 501.034,A -85,B 0,C 180,E1 -16973.684,E2 -16973.684} C_VEL
LIN {X 0,Y 303.63,Z 511.888,A -85,B 0,C 180,E1 -16975.986,E2 -16975.986} C_VEL
LIN {X 0,Y 303.373,Z 521.786,A -85,B 0,C 180,E1 -16977.804,E2 -16977.804} C_VEL
LIN {X 0,Y 302.239,Z 532.89,A -85,B 0,C 180,E1 -16979.665,E2 -16979.665} C_VEL
LIN {X 0,Y 299.482,Z 547.134,A -85,B 0,C 180,E1 -16982.008,E2 -16982.008} C_VEL
LIN {X 0,Y 297.971,Z 555.567,A -85,B 0,C 180,E1 -16983.581,E2 -16983.581} C_VEL
LIN {X 0,Y 295.004,Z 564.492,A -85,B 0,C 180,E1 -16985.189,E2 -16985.189} C_VEL
LIN {X 0,Y 292.721,Z 576.302,A -85,B 0,C 180,E1 -16986.849,E2 -16986.849} C_VEL
LIN {X 0,Y 290.471,Z 587.043,A -85,B 0,C 180,E1 -16988.72,E2 -16988.72} C_VEL
LIN {X 0,Y 288.383,Z 596.705,A -85,B 0,C 180,E1 -16990.792,E2 -16990.792} C_VEL
LIN {X 0,Y 286.547,Z 605.242,A -85,B 0,C 180,E1 -16993.045,E2 -16993.045} C_VEL
LIN {X 0,Y 285.35,Z 611.344,A -85,B 0,C 180,E1 -16995.012,E2 -16995.012} C_VEL
LIN {X 0,Y 284.119,Z 616.85,A -85,B 0,C 180,E1 -16997.137,E2 -16997.137} C_VEL
LIN {X 0,Y 283.141,Z 622.608,A -85,B 0,C 180,E1 -16999.994,E2 -16999.994} C_VEL
LIN {X 0,Y 282.598,Z 626.786,A -85,B 0,C 180,E1 -17002.857,E2 -17002.857} C_VEL
LIN {X 0,Y 282.378,Z 629.514,A -85,B 0,C 180,E1 -17005.718,E2 -17005.718} C_VEL
LIN {X 0,Y 282.36,Z 630.869,A -85,B 0,C 180,E1 -17008.574,E2 -17008.574} C_VEL
LIN {X 0,Y 282.36,Z 630.864,A -85,B 0,C 180,E1 -17011.426,E2 -17011.426} C_VEL
LIN {X 0,Y 282.369,Z 629.504,A -85,B 0,C 180,E1 -17014.282,E2 -17014.282} C_VEL
LIN {X 0,Y 282.591,Z 626.769,A -85,B 0,C 180,E1 -17017.143,E2 -17017.143} C_VEL
LIN {X 0,Y 283.129,Z 622.578,A -85,B 0,C 180,E1 -17020.006,E2 -17020.006} C_VEL
LIN {X 0,Y 284.11,Z 616.809,A -85,B 0,C 180,E1 -17022.864,E2 -17022.864} C_VEL
LIN {X 0,Y 285.444,Z 610.289,A -85,B 0,C 180,E1 -17025.348,E2 -17025.348} C_VEL
LIN {X 0,Y 287.135,Z 602.168,A -85,B 0,C 180,E1 -17027.816,E2 -17027.816} C_VEL
LIN {X 0,Y 289.007,Z 593.645,A -85,B 0,C 180,E1 -17029.904,E2 -17029.904} C_VEL
LIN {X 0,Y 291.199,Z 583.29,A -85,B 0,C 180,E1 -17031.968,E2 -17031.968} C_VEL
LIN {X 0,Y 293.387,Z 572.858,A -85,B 0,C 180,E1 -17033.656,E2 -17033.656} C_VEL
LIN {X 0,Y 295.516,Z 561.204,A -85,B 0,C 180,E1 -17035.195,E2 -17035.195} C_VEL
LIN {X 0,Y 296.823,Z 552.455,A -85,B 0,C 180,E1 -17036.167,E2 -17036.167} C_VEL
LIN {X 0,Y 296.082,Z 539.741,A -85,B 0,C 180,E1 -17037.547,E2 -17037.547} C_VEL
LIN {X 0,Y 294.483,Z 525.839,A -85,B 0,C 180,E1 -17038.813,E2 -17038.813} C_VEL
LIN {X 0,Y 292.291,Z 511.226,A -85,B 0,C 180,E1 -17039.877,E2 -17039.877} C_VEL
LIN {X 0,Y 290.298,Z 502.751,A -85,B 0,C 180,E1 -17040.433,E2 -17040.433} C_VEL
LIN {X 0,Y 286.307,Z 489.975,A -85,B 0,C 180,E1 -17041.291,E2 -17041.291} C_VEL
LIN {X 0,Y 284.794,Z 477.927,A -85,B 0,C 180,E1 -17043.567,E2 -17043.567} C_VEL
LIN {X 0,Y 285.284,Z 472.304,A -85,B 0,C 180,E1 -17047.125,E2 -17047.125} C_VEL
LIN {X 0,Y 285.846,Z 467.309,A -85,B 0,C 180,E1 -17050.343,E2 -17050.343} C_VEL
LIN {X 0,Y 286.645,Z 460.676,A -85,B 0,C 180,E1 -17054.682,E2 -17054.682} C_VEL
LIN {X 0,Y 287.02,Z 456.829,A -85,B 0,C 180,E1 -17057.272,E2 -17057.272} C_VEL
LIN {X 0,Y 286.939,Z 453.781,A -85,B 0,C 180,E1 -17059.401,E2 -17059.401} C_VEL
LIN {X 0,Y 286.09,Z 448.829,A -85,B 0,C 180,E1 -17062.997,E2 -17062.997} C_VEL
LIN {X 0,Y 285.212,Z 443.319,A -85,B 0,C 180,E1 -17067.173,E2 -17067.173} C_VEL
LIN {X 0,Y 284.391,Z 438.689,A -85,B 0,C 180,E1 -17070.989,E2 -17070.989} C_VEL
LIN {X 0,Y 284.379,Z 438.668,A -85,B 0,C 180,E1 -17073.587,E2 -17073.587} C_VEL
LIN {X 0,Y 284.368,Z 438.689,A -85,B 0,C 180,E1 -17076.707,E2 -17076.707} C_VEL
LIN {X 0,Y 284.406,Z 438.679,A -85,B 0,C 180,E1 -17081.262,E2 -17081.262} C_VEL
LIN {X 0,Y 284.493,Z 438.653,A -85,B 0,C 180,E1 -17084.459,E2 -17084.459} C_VEL
LIN {X 0,Y 284.484,Z 438.673,A -85,B 0,C 180,E1 -17088.601,E2 -17088.601} C_VEL
LIN {X 0,Y 284.602,Z 438.637,A -85,B 0,C 180,E1 -17091.48,E2 -17091.48} C_VEL
LIN {X 0,Y 284.596,Z 438.66,A -85,B 0,C 180,E1 -17094.331,E2 -17094.331} C_VEL
LIN {X 0,Y 284.857,Z 438.617,A -85,B 0,C 180,E1 -17098.586,E2 -17098.586} C_VEL
LIN {X 0,Y 284.857,Z 438.618,A -85,B 0,C 180,E1 -17101.414,E2 -17101.414} C_VEL
LIN {X 0,Y 284.7,Z 438.638,A -85,B 0,C 180,E1 -17107.09,E2 -17107.09} C_VEL
LIN {X 0,Y 284.568,Z 438.653,A -85,B 0,C 180,E1 -17109.955,E2 -17109.955} C_VEL
LIN {X 0,Y 284.483,Z 438.659,A -85,B 0,C 180,E1 -17114.303,E2 -17114.303} C_VEL
LIN {X 0,Y 284.425,Z 438.677,A -85,B 0,C 180,E1 -17117.249,E2 -17117.249} C_VEL
LIN {X 0,Y 284.379,Z 438.686,A -85,B 0,C 180,E1 -17120.242,E2 -17120.242} C_VEL
LIN {X 0,Y 284.34,Z 438.693,A -85,B 0,C 180,E1 -17124.847,E2 -17124.847} C_VEL
LIN {X 0,Y 284.334,Z 438.691,A -85,B 0,C 180,E1 -17128.011,E2 -17128.011} C_VEL
LIN {X 0,Y 284.297,Z 438.697,A -85,B 0,C 180,E1 -17131.274,E2 -17131.274} C_VEL
LIN {X 0,Y 284.339,Z 438.815,A -85,B 0,C 180,E1 -17134.86,E2 -17134.86} C_VEL
LIN {X 0,Y 286.234,Z 446.108,A -85,B 0,C 180,E1 -17138.763,E2 -17138.763} C_VEL
LIN {X 0,Y 288.088,Z 454.398,A -85,B 0,C 180,E1 -17142.957,E2 -17142.957} C_VEL
LIN {X 0,Y 289.69,Z 463.171,A -85,B 0,C 180,E1 -17147.212,E2 -17147.212} C_VEL
LIN {X 0,Y 290.096,Z 468.463,A -85,B 0,C 180,E1 -17149.605,E2 -17149.605} C_VEL
LIN {X 0,Y 289.027,Z 478.591,A -85,B 0,C 180,E1 -17153.808,E2 -17153.808} C_VEL
LIN {X 0,Y 288.115,Z 489.673,A -85,B 0,C 180,E1 -17158.222,E2 -17158.222} C_VEL
LIN {X 0,Y 287.973,Z 491.462,A -85,B 0,C 180,E1 -17158.868,E2 -17158.868} C_VEL
LIN {X 0,Y 292.761,Z 507.528,A -85,B 0,C 180,E1 -17160.008,E2 -17160.008} C_VEL
LIN {X 0,Y 295.892,Z 521.467,A -85,B 0,C 180,E1 -17161.164,E2 -17161.164} C_VEL
LIN {X 0,Y 297.986,Z 535.417,A -85,B 0,C 180,E1 -17162.502,E2 -17162.502} C_VEL
LIN {X 0,Y 298.481,Z 541.381,A -85,B 0,C 180,E1 -17163.134,E2 -17163.134} C_VEL
LIN {X 0,Y 296.661,Z 554.421,A -85,B 0,C 180,E1 -17164.48,E2 -17164.48} C_VEL
LIN {X 0,Y 294.373,Z 566.679,A -85,B 0,C 180,E1 -17166.055,E2 -17166.055} C_VEL
LIN {X 0,Y 292.11,Z 577.291,A -85,B 0,C 180,E1 -17167.732,E2 -17167.732} C_VEL
LIN {X 0,Y 289.842,Z 587.795,A -85,B 0,C 180,E1 -17169.786,E2 -17169.786} C_VEL
LIN {X 0,Y 287.811,Z 596.467,A -85,B 0,C 180,E1 -17171.86,E2 -17171.86} C_VEL
LIN {X 0,Y 286.388,Z 603.67,A -85,B 0,C 180,E1 -17173.974,E2 -17173.974} C_VEL
LIN {X 0,Y 284.793,Z 610.554,A -85,B 0,C 180,E1 -17176.442,E2 -17176.442} C_VEL
LIN {X 0,Y 283.546,Z 616.723,A -85,B 0,C 180,E1 -17179.287,E2 -17179.287} C_VEL
LIN {X 0,Y 282.958,Z 620.23,A -85,B 0,C 180,E1 -17181.43,E2 -17181.43} C_VEL
LIN {X 0,Y 282.481,Z 623.739,A -85,B 0,C 180,E1 -17184.377,E2 -17184.377} C_VEL
LIN {X 0,Y 282.349,Z 625.682,A -85,B 0,C 180,E1 -17187.146,E2 -17187.146} C_VEL
LIN {X 0,Y 282.295,Z 626.379,A -85,B 0,C 180,E1 -17190,E2 -17190} C_VEL
LIN {X 0,Y 282.347,Z 625.741,A -85,B 0,C 180,E1 -17192.854,E2 -17192.854} C_VEL
LIN {X 0,Y 282.483,Z 623.759,A -85,B 0,C 180,E1 -17195.711,E2 -17195.711} C_VEL
LIN {X 0,Y 282.956,Z 620.391,A -85,B 0,C 180,E1 -17198.571,E2 -17198.571} C_VEL
LIN {X 0,Y 283.782,Z 615.538,A -85,B 0,C 180,E1 -17201.427,E2 -17201.427} C_VEL
LIN {X 0,Y 284.738,Z 610.832,A -85,B 0,C 180,E1 -17203.561,E2 -17203.561} C_VEL
LIN {X 0,Y 286.301,Z 604.009,A -85,B 0,C 180,E1 -17206.031,E2 -17206.031} C_VEL
LIN {X 0,Y 288.125,Z 595.542,A -85,B 0,C 180,E1 -17208.488,E2 -17208.488} C_VEL
LIN {X 0,Y 290.166,Z 586.685,A -85,B 0,C 180,E1 -17210.561,E2 -17210.561} C_VEL
LIN {X 0,Y 292.418,Z 575.962,A -85,B 0,C 180,E1 -17212.616,E2 -17212.616} C_VEL
LIN {X 0,Y 294.759,Z 565.079,A -85,B 0,C 180,E1 -17214.286,E2 -17214.286} C_VEL
LIN {X 0,Y 296.859,Z 553.212,A -85,B 0,C 180,E1 -17215.773,E2 -17215.773} C_VEL
LIN {X 0,Y 298.501,Z 542.31,A -85,B 0,C 180,E1 -17216.882,E2 -17216.882} C_VEL
LIN {X 0,Y 297.65,Z 532.558,A -85,B 0,C 180,E1 -17217.899,E2 -17217.899} C_VEL
LIN {X 0,Y 295.472,Z 519.209,A -85,B 0,C 180,E1 -17219.15,E2 -17219.15} C_VEL
LIN {X 0,Y 292.171,Z 505.193,A -85,B 0,C 180,E1 -17220.286,E2 -17220.286} C_VEL
LIN {X 0,Y 287.964,Z 491.283,A -85,B 0,C 180,E1 -17221.279,E2 -17221.279} C_VEL
LIN {X 0,Y 288.829,Z 481.129,A -85,B 0,C 180,E1 -17225.303,E2 -17225.303} C_VEL
LIN {X 0,Y 289.853,Z 470.832,A -85,B 0,C 180,E1 -17229.53,E2 -17229.53} C_VEL
LIN {X 0,Y 290.078,Z 466.647,A -85,B 0,C 180,E1 -17231.317,E2 -17231.317} C_VEL
LIN {X 0,Y 289.227,Z 460.499,A -85,B 0,C 180,E1 -17234.196,E2 -17234.196} C_VEL
LIN {X 0,Y 287.804,Z 453.11,A -85,B 0,C 180,E1 -17237.867,E2 -17237.867} C_VEL
LIN {X 0,Y 285.945,Z 444.8,A -85,B 0,C 180,E1 -17242.088,E2 -17242.088} C_VEL
LIN {X 0,Y 284.315,Z 438.686,A -85,B 0,C 180,E1 -17245.459,E2 -17245.459} C_VEL
LIN {X 0,Y 284.318,Z 438.68,A -85,B 0,C 180,E1 -17249.901,E2 -17249.901} C_VEL
LIN {X 0,Y 284.343,Z 438.678,A -85,B 0,C 180,E1 -17250.2,E2 -17250.2} C_VEL
LIN {X 0,Y 289.216,Z 453.501,A -85,B 0,C 180,E1 -17251.829,E2 -17251.829} C_VEL
LIN {X 0,Y 293.55,Z 467.793,A -85,B 0,C 180,E1 -17253.639,E2 -17253.639} C_VEL
LIN {X 0,Y 294.754,Z 472.472,A -85,B 0,C 180,E1 -17254.285,E2 -17254.285} C_VEL
LIN {X 0,Y 292.952,Z 485.504,A -85,B 0,C 180,E1 -17255.931,E2 -17255.931} C_VEL
LIN {X 0,Y 291.106,Z 498.072,A -85,B 0,C 180,E1 -17257.838,E2 -17257.838} C_VEL
LIN {X 0,Y 289.522,Z 508.711,A -85,B 0,C 180,E1 -17259.762,E2 -17259.762} C_VEL
LIN {X 0,Y 289.139,Z 511.234,A -85,B 0,C 180,E1 -17260.265,E2 -17260.265} C_VEL
LIN {X 0,Y 287.869,Z 515.304,A -85,B 0,C 180,E1 -17261.087,E2 -17261.087} C_VEL
LIN {X 0,Y 284.203,Z 521.623,A -85,B 0,C 180,E1 -17262.415,E2 -17262.415} C_VEL
LIN {X 0,Y 280.534,Z 527.598,A -85,B 0,C 180,E1 -17263.838,E2 -17263.838} C_VEL
LIN {X 0,Y 279.286,Z 530.981,A -85,B 0,C 180,E1 -17264.798,E2 -17264.798} C_VEL
LIN {X 0,Y 278.034,Z 539.462,A -85,B 0,C 180,E1 -17267.593,E2 -17267.593} C_VEL
LIN {X 0,Y 277.208,Z 546.605,A -85,B 0,C 180,E1 -17270.515,E2 -17270.515} C_VEL
LIN {X 0,Y 276.699,Z 552.208,A -85,B 0,C 180,E1 -17273.437,E2 -17273.437} C_VEL
LIN {X 0,Y 276.636,Z 555.52,A -85,B 0,C 180,E1 -17275.629,E2 -17275.629} C_VEL
LIN {X 0,Y 276.348,Z 558.794,A -85,B 0,C 180,E1 -17278.543,E2 -17278.543} C_VEL
LIN {X 0,Y 276.411,Z 560.844,A -85,B 0,C 180,E1 -17281.457,E2 -17281.457} C_VEL
LIN {X 0,Y 276.999,Z 561.681,A -85,B 0,C 180,E1 -17284.365,E2 -17284.365} C_VEL
LIN {X 0,Y 278.022,Z 561.336,A -85,B 0,C 180,E1 -17287.261,E2 -17287.261} C_VEL
LIN {X 0,Y 279.295,Z 559.846,A -85,B 0,C 180,E1 -17290.145,E2 -17290.145} C_VEL
LIN {X 0,Y 280.933,Z 557.211,A -85,B 0,C 180,E1 -17293.012,E2 -17293.012} C_VEL
LIN {X 0,Y 282.971,Z 553.36,A -85,B 0,C 180,E1 -17295.855,E2 -17295.855} C_VEL
LIN {X 0,Y 285.742,Z 548.176,A -85,B 0,C 180,E1 -17298.647,E2 -17298.647} C_VEL
LIN {X 0,Y 288.161,Z 543.392,A -85,B 0,C 180,E1 -17300.71,E2 -17300.71} C_VEL
LIN {X 0,Y 291.609,Z 536.3,A -85,B 0,C 180,E1 -17303.199,E2 -17303.199} C_VEL
LIN {X 0,Y 295.607,Z 527.505,A -85,B 0,C 180,E1 -17305.715,E2 -17305.715} C_VEL
LIN {X 0,Y 299.749,Z 517.804,A -85,B 0,C 180,E1 -17307.964,E2 -17307.964} C_VEL
LIN {X 0,Y 303.75,Z 508.023,A -85,B 0,C 180,E1 -17309.832,E2 -17309.832} C_VEL
LIN {X 0,Y 308.461,Z 495.394,A -85,B 0,C 180,E1 -17311.852,E2 -17311.852} C_VEL
LIN {X 0,Y 307.971,Z 490.876,A -85,B 0,C 180,E1 -17313.209,E2 -17313.209} C_VEL
LIN {X 0,Y 306.751,Z 484.836,A -85,B 0,C 180,E1 -17315.378,E2 -17315.378} C_VEL
LIN {X 0,Y 305.726,Z 482.147,A -85,B 0,C 180,E1 -17316.704,E2 -17316.704} C_VEL
LIN {X 0,Y 303.786,Z 480.139,A -85,B 0,C 180,E1 -17318.655,E2 -17318.655} C_VEL
LIN {X 0,Y 302.139,Z 479.476,A -85,B 0,C 180,E1 -17320.64,E2 -17320.64} C_VEL
LIN {X 0,Y 301.402,Z 479.462,A -85,B 0,C 180,E1 -17321.74,E2 -17321.74} C_VEL
LIN {X 0,Y 300.35,Z 480.622,A -85,B 0,C 180,E1 -17323.499,E2 -17323.499} C_VEL
LIN {X 0,Y 299.512,Z 482.987,A -85,B 0,C 180,E1 -17325.256,E2 -17325.256} C_VEL
LIN {X 0,Y 298.449,Z 489.271,A -85,B 0,C 180,E1 -17327.965,E2 -17327.965} C_VEL
LIN {X 0,Y 298.531,Z 493.62,A -85,B 0,C 180,E1 -17329.714,E2 -17329.714} C_VEL
LIN {X 0,Y 298.592,Z 500.961,A -85,B 0,C 180,E1 -17331.89,E2 -17331.89} C_VEL
LIN {X 0,Y 298.666,Z 505.784,A -85,B 0,C 180,E1 -17333.136,E2 -17333.136} C_VEL
LIN {X 0,Y 298.59,Z 516.232,A -85,B 0,C 180,E1 -17335.467,E2 -17335.467} C_VEL
LIN {X 0,Y 297.858,Z 526.04,A -85,B 0,C 180,E1 -17337.354,E2 -17337.354} C_VEL
LIN {X 0,Y 296.466,Z 535.498,A -85,B 0,C 180,E1 -17339.039,E2 -17339.039} C_VEL
LIN {X 0,Y 293.064,Z 550.705,A -85,B 0,C 180,E1 -17341.73,E2 -17341.73} C_VEL
LIN {X 0,Y 292.091,Z 555.975,A -85,B 0,C 180,E1 -17342.796,E2 -17342.796} C_VEL
LIN {X 0,Y 288.088,Z 566.958,A -85,B 0,C 180,E1 -17344.928,E2 -17344.928} C_VEL
LIN {X 0,Y 285.765,Z 578.386,A -85,B 0,C 180,E1 -17346.636,E2 -17346.636} C_VEL
LIN {X 0,Y 283.457,Z 588.769,A -85,B 0,C 180,E1 -17348.549,E2 -17348.549} C_VEL
LIN {X 0,Y 281.303,Z 598.127,A -85,B 0,C 180,E1 -17350.668,E2 -17350.668} C_VEL
LIN {X 0,Y 279.449,Z 606.679,A -85,B 0,C 180,E1 -17353.077,E2 -17353.077} C_VEL
LIN {X 0,Y 278.032,Z 613.27,A -85,B 0,C 180,E1 -17355.358,E2 -17355.358} C_VEL
LIN {X 0,Y 276.842,Z 618.404,A -85,B 0,C 180,E1 -17357.539,E2 -17357.539} C_VEL
LIN {X 0,Y 276.128,Z 622.551,A -85,B 0,C 180,E1 -17359.737,E2 -17359.737} C_VEL
LIN {X 0,Y 275.525,Z 626.728,A -85,B 0,C 180,E1 -17362.673,E2 -17362.673} C_VEL
LIN {X 0,Y 275.287,Z 629.456,A -85,B 0,C 180,E1 -17365.607,E2 -17365.607} C_VEL
LIN {X 0,Y 275.284,Z 630.81,A -85,B 0,C 180,E1 -17368.537,E2 -17368.537} C_VEL
LIN {X 0,Y 275.284,Z 630.806,A -85,B 0,C 180,E1 -17371.463,E2 -17371.463} C_VEL
LIN {X 0,Y 275.28,Z 629.445,A -85,B 0,C 180,E1 -17374.393,E2 -17374.393} C_VEL
LIN {X 0,Y 275.516,Z 626.71,A -85,B 0,C 180,E1 -17377.328,E2 -17377.328} C_VEL
LIN {X 0,Y 276.117,Z 622.52,A -85,B 0,C 180,E1 -17380.263,E2 -17380.263} C_VEL
LIN {X 0,Y 277.17,Z 616.751,A -85,B 0,C 180,E1 -17383.192,E2 -17383.192} C_VEL
LIN {X 0,Y 278.556,Z 610.231,A -85,B 0,C 180,E1 -17385.737,E2 -17385.737} C_VEL
LIN {X 0,Y 280.348,Z 602.111,A -85,B 0,C 180,E1 -17388.262,E2 -17388.262} C_VEL
LIN {X 0,Y 282.306,Z 593.59,A -85,B 0,C 180,E1 -17390.397,E2 -17390.397} C_VEL
LIN {X 0,Y 284.608,Z 583.237,A -85,B 0,C 180,E1 -17392.504,E2 -17392.504} C_VEL
LIN {X 0,Y 286.876,Z 572.807,A -85,B 0,C 180,E1 -17394.227,E2 -17394.227} C_VEL
LIN {X 0,Y 289.064,Z 561.156,A -85,B 0,C 180,E1 -17395.798,E2 -17395.798} C_VEL
LIN {X 0,Y 290.295,Z 552.41,A -85,B 0,C 180,E1 -17396.801,E2 -17396.801} C_VEL
LIN {X 0,Y 289.55,Z 539.703,A -85,B 0,C 180,E1 -17398.223,E2 -17398.223} C_VEL
LIN {X 0,Y 287.982,Z 525.739,A -85,B 0,C 180,E1 -17399.532,E2 -17399.532} C_VEL
LIN {X 0,Y 285.853,Z 511.116,A -85,B 0,C 180,E1 -17400.626,E2 -17400.626} C_VEL
LIN {X 0,Y 282.15,Z 497.751,A -85,B 0,C 180,E1 -17401.57,E2 -17401.57} C_VEL
LIN {X 0,Y 279.591,Z 490.023,A -85,B 0,C 180,E1 -17402.133,E2 -17402.133} C_VEL
LIN {X 0,Y 278.267,Z 479.691,A -85,B 0,C 180,E1 -17404.191,E2 -17404.191} C_VEL
LIN {X 0,Y 277.895,Z 476.161,A -85,B 0,C 180,E1 -17404.903,E2 -17404.903} C_VEL
LIN {X 0,Y 278.547,Z 469.73,A -85,B 0,C 180,E1 -17409.107,E2 -17409.107} C_VEL
LIN {X 0,Y 279.249,Z 463.683,A -85,B 0,C 180,E1 -17413.126,E2 -17413.126} C_VEL
LIN {X 0,Y 279.909,Z 458.419,A -85,B 0,C 180,E1 -17416.73,E2 -17416.73} C_VEL
LIN {X 0,Y 279.908,Z 454.834,A -85,B 0,C 180,E1 -17419.246,E2 -17419.246} C_VEL
LIN {X 0,Y 279.111,Z 450.032,A -85,B 0,C 180,E1 -17422.82,E2 -17422.82} C_VEL
LIN {X 0,Y 278.306,Z 445.313,A -85,B 0,C 180,E1 -17426.444,E2 -17426.444} C_VEL
LIN {X 0,Y 277.537,Z 440.408,A -85,B 0,C 180,E1 -17430.41,E2 -17430.41} C_VEL
LIN {X 0,Y 277.342,Z 439.567,A -85,B 0,C 180,E1 -17431.219,E2 -17431.219} C_VEL
LIN {X 0,Y 277.315,Z 439.548,A -85,B 0,C 180,E1 -17434.48,E2 -17434.48} C_VEL
LIN {X 0,Y 277.287,Z 439.565,A -85,B 0,C 180,E1 -17437.655,E2 -17437.655} C_VEL
LIN {X 0,Y 277.347,Z 439.551,A -85,B 0,C 180,E1 -17440.766,E2 -17440.766} C_VEL
LIN {X 0,Y 277.436,Z 439.529,A -85,B 0,C 180,E1 -17445.326,E2 -17445.326} C_VEL
LIN {X 0,Y 277.459,Z 439.534,A -85,B 0,C 180,E1 -17449.787,E2 -17449.787} C_VEL
LIN {X 0,Y 277.625,Z 439.518,A -85,B 0,C 180,E1 -17452.728,E2 -17452.728} C_VEL
LIN {X 0,Y 277.823,Z 439.492,A -85,B 0,C 180,E1 -17458.551,E2 -17458.551} C_VEL
LIN {X 0,Y 277.823,Z 439.494,A -85,B 0,C 180,E1 -17461.45,E2 -17461.45} C_VEL
LIN {X 0,Y 277.655,Z 439.513,A -85,B 0,C 180,E1 -17467.271,E2 -17467.271} C_VEL
LIN {X 0,Y 277.508,Z 439.536,A -85,B 0,C 180,E1 -17470.211,E2 -17470.211} C_VEL
LIN {X 0,Y 277.436,Z 439.538,A -85,B 0,C 180,E1 -17474.674,E2 -17474.674} C_VEL
LIN {X 0,Y 277.344,Z 439.551,A -85,B 0,C 180,E1 -17479.234,E2 -17479.234} C_VEL
LIN {X 0,Y 277.294,Z 439.565,A -85,B 0,C 180,E1 -17484.158,E2 -17484.158} C_VEL
LIN {X 0,Y 277.328,Z 439.558,A -85,B 0,C 180,E1 -17487.505,E2 -17487.505} C_VEL
LIN {X 0,Y 277.273,Z 439.565,A -85,B 0,C 180,E1 -17490.481,E2 -17490.481} C_VEL
LIN {X 0,Y 277.258,Z 439.672,A -85,B 0,C 180,E1 -17493.675,E2 -17493.675} C_VEL
LIN {X 0,Y 278.966,Z 445.963,A -85,B 0,C 180,E1 -17497.203,E2 -17497.203} C_VEL
LIN {X 0,Y 280.476,Z 452.47,A -85,B 0,C 180,E1 -17500.655,E2 -17500.655} C_VEL
LIN {X 0,Y 281.689,Z 458.338,A -85,B 0,C 180,E1 -17503.653,E2 -17503.653} C_VEL
LIN {X 0,Y 282.929,Z 465.151,A -85,B 0,C 180,E1 -17507.024,E2 -17507.024} C_VEL
LIN {X 0,Y 283.379,Z 469.415,A -85,B 0,C 180,E1 -17509.004,E2 -17509.004} C_VEL
LIN {X 0,Y 282.425,Z 478.359,A -85,B 0,C 180,E1 -17512.779,E2 -17512.779} C_VEL
